	W =   -44.397 deg,	P =     8.168 deg,	R =    14.048 deg
   GP2:
	UF : 1, UT : 1,
	J1=    90.000 deg,	J2=   -90.000 deg
};
P[588]{
   GP1:
	UF : 1, UT : 1,		CONFIG : 'N U T, 0, 0, 0',
	X =  2413.075  mm,	Y =    96.166  mm,	Z =    -3.839  mm,
	W =   -44.394 deg,	P =     8.166 deg,	R =    14.048 deg
   GP2:
	UF : 1, UT : 1,
	J1=    90.000 deg,	J2=   -90.000 deg
};
P[589]{
   GP1:
	UF : 1, UT : 1,		CONFIG : 'N U T, 0, 0, 0',
	X =  1890.253  mm,	Y =  -197.333  mm,	Z =   104.046  mm,
	W =    40.690 deg,	P =   -21.162 deg,	R =    -6.795 deg
   GP2:
	UF : 1, UT : 1,
	J1=    90.000 deg,	J2=   -90.000 deg
};
P[590]{
   GP1:
	UF : 1, UT : 1,		CONFIG : 'N U T, 0, 0, 0',
	X =  1890.254  mm,	Y =  -197.333  mm,	Z =   104.046  mm,
	W =   -33.760 deg,	P =   -16.746 deg,	R =    41.760 deg
   GP2:
	UF : 1, UT : 1,
	J1=    90.000 deg,	J2=   -90.000 deg
};
P[591]{
   GP1:
	UF : 1, UT : 1,		CONFIG : 'N U T, 0, 0, 0',
	X =  2024.254  mm,	Y =  -116.333  mm,	Z =   104.046  mm,
	W =   -36.632 deg,	P =    -7.222 deg,	R =    55.482 deg
   GP2:
	UF : 1, UT : 1,
	J1=    90.000 deg,	J2=   -90.000 deg
};
P[592]{
   GP1:
	UF : 1, UT : 1,		CONFIG : 'N U T, 0, 0, 0',
	X =  2427.383  mm,	Y =    97.382  mm,	Z =     -.048  mm,
	W =   -44.529 deg,	P =    -7.125 deg,	R =    33.229 deg
   GP2:
	UF : 1, UT : 1,
	J1=    90.000 deg,	J2=   -90.000 deg
};
P[593]{
   GP1:
	UF : 1, UT : 1,		CONFIG : 'N U T, 0, 0, 0',
	X =  2337.427  mm,	Y =    71.440  mm,	Z =   847.749  mm,
	W =    45.399 deg,	P =    17.266 deg,	R =    -1.541 deg
   GP2:
	UF : 1, UT : 1,
	J1=    90.000 deg,	J2=   -90.000 deg
};
P[594]{
   GP1:
	UF : 1, UT : 1,		CONFIG : 'N U T, 0, 0, 0',
	X =  2402.831  mm,	Y =   104.785  mm,	Z =   847.602  mm,
	W =    45.390 deg,	P =    17.268 deg,	R =    -1.529 deg
   GP2:
	UF : 1, UT : 1,
	J1=    90.000 deg,	J2=   -90.000 deg
};
P[595]{
   GP1:
	UF : 1, UT : 1,		CONFIG : 'N U T, 0, 0, 0',
	X =  2056.301  mm,	Y =   -98.366  mm,	Z =    49.506  mm,
	W =   -42.382 deg,	P =     2.305 deg,	R =   105.198 deg
   GP2:
	UF : 1, UT : 1,
	J1=    90.000 deg,	J2=   -90.000 deg
};
P[596]{
   GP1:
	UF : 1, UT : 1,		CONFIG : 'N U T, 0, 0, 1',
	X =  1663.323  mm,	Y =  -387.368  mm,	Z =   408.939  mm,
	W =   -27.547 deg,	P =    30.353 deg,	R =   152.229 deg
   GP2:
	UF : 1, UT : 1,
	J1=    90.000 deg,	J2=   -90.000 deg
};
P[597]{
   GP1:
	UF : 1, UT : 1,		CONFIG : 'N U T, 0, 0, 1',
	X =  1656.330  mm,	Y =  -300.541  mm,	Z =  1123.310  mm,
	W =    -7.423 deg,	P =    33.575 deg,	R =  -172.195 deg
   GP2:
	UF : 1, UT : 1,
	J1=    90.000 deg,	J2=   -90.000 deg
};
P[598]{
   GP1:
	UF : 1, UT : 1,		CONFIG : 'N U T, 0, 0, 1',
	X =  2106.086  mm,	Y =  -147.825  mm,	Z =   986.847  mm,
	W =    -2.744 deg,	P =    30.268 deg,	R =  -167.022 deg
   GP2:
	UF : 1, UT : 1,
	J1=    90.000 deg,	J2=   -90.000 deg
};
P[599]{
   GP1:
	UF : 1, UT : 1,		CONFIG : 'N U T, 0, 0, 0',
	X =  2402.842  mm,	Y =   109.949  mm,	Z =   847.942  mm,
	W =     1.452 deg,	P =    40.371 deg,	R =    26.792 deg
   GP2:
	UF : 1, UT : 1,
	J1=    90.000 deg,	J2=   -90.000 deg
};
P[600]{
   GP1:
	UF : 1, UT : 1,		CONFIG : 'N U T, 0, 0, 0',
	X =  2392.403  mm,	Y =   126.094  mm,	Z =   845.932  mm,
	W =     1.448 deg,	P =    40.368 deg,	R =    26.765 deg
   GP2:
	UF : 1, UT : 1,
	J1=    90.000 deg,	J2=   -90.000 deg
};
P[601]{
   GP1:
	UF : 1, UT : 1,		CONFIG : 'F U T, 0, 0, 0',
	X =  2325.472  mm,	Y =    92.116  mm,	Z =   847.036  mm,
	W =   -46.230 deg,	P =   -25.147 deg,	R =    34.050 deg
   GP2:
	UF : 1, UT : 1,
	J1=    90.000 deg,	J2=   -90.000 deg
};
P[602]{
   GP1:
	UF : 1, UT : 1,		CONFIG : 'F U T, 0, 0, 0',
	X =  2391.645  mm,	Y =   126.896  mm,	Z =   847.777  mm,
	W =   -46.222 deg,	P =   -25.150 deg,	R =    34.042 deg
   GP2:
	UF : 1, UT : 1,
	J1=    90.000 deg,	J2=   -90.000 deg
};
P[603]{
   GP1:
	UF : 1, UT : 1,		CONFIG : 'N U T, 0, 0, 0',
	X =  2011.750  mm,	Y =   -80.950  mm,	Z =    -4.575  mm,
	W =    40.372 deg,	P =    23.935 deg,	R =    74.339 deg
   GP2:
	UF : 1, UT : 1,
	J1=    90.000 deg,	J2=  -100.000 deg
};
P[604]{
   GP1:
	UF : 1, UT : 1,		CONFIG : 'N U T, 0, 0, 0',
	X =  2007.194  mm,	Y =   142.177  mm,	Z =   -45.001  mm,
	W =    45.685 deg,	P =     4.509 deg,	R =    78.826 deg
   GP2:
	UF : 1, UT : 1,
	J1=    90.000 deg,	J2=  -100.000 deg
};
P[605]{
   GP1:
	UF : 1, UT : 1,		CONFIG : 'N U T, 0, 0, 0',
	X =  2229.070  mm,	Y =   -48.871  mm,	Z =     4.516  mm,
	W =    44.904 deg,	P =    -3.411 deg,	R =     3.413 deg
   GP2:
	UF : 1, UT : 1,
	J1=    90.000 deg,	J2=   -90.000 deg
};
P[606]{
   GP1:
	UF : 1, UT : 1,		CONFIG : 'N U T, 0, 0, 0',
	X =  2266.341  mm,	Y =   -46.762  mm,	Z =     3.253  mm,
	W =    44.893 deg,	P =    -3.421 deg,	R =     3.427 deg
   GP2:
	UF : 1, UT : 1,
	J1=    90.000 deg,	J2=   -90.000 deg
};
P[607]{
   GP1:
	UF : 1, UT : 1,		CONFIG : 'N U T, 0, 0, 0',
	X =  2096.605  mm,	Y =  -181.583  mm,	Z =   897.867  mm,
	W =     -.064 deg,	P =    31.734 deg,	R =  -164.129 deg
   GP2:
	UF : 1, UT : 1,
	J1=    90.000 deg,	J2=   -90.000 deg
};
P[608]{
   GP1:
	UF : 1, UT : 1,		CONFIG : 'N U T, 0, 0, 0',
	X =  2114.149  mm,	Y =  -253.336  mm,	Z =   921.197  mm,
	W =     1.157 deg,	P =    35.359 deg,	R =   -90.786 deg
   GP2:
	UF : 1, UT : 1,
	J1=    90.000 deg,	J2=   -90.000 deg
};
P[609]{
   GP1:
	UF : 1, UT : 1,		CONFIG : 'N U T, 0, 0, 0',
	X =  2142.334  mm,	Y =   -48.860  mm,	Z =    -3.830  mm,
	W =    44.883 deg,	P =     3.632 deg,	R =    -4.928 deg
   GP2:
	UF : 1, UT : 1,
	J1=    90.000 deg,	J2=   -90.000 deg
};
P[610]{
   GP1:
	UF : 1, UT : 1,		CONFIG : 'N U T, 0, 0, 0',
	X =  2212.734  mm,	Y =   -47.597  mm,	Z =    -4.519  mm,
	W =    44.886 deg,	P =     3.634 deg,	R =    -4.918 deg
   GP2:
	UF : 1, UT : 1,
	J1=    90.000 deg,	J2=   -90.000 deg
};
P[611]{
   GP1:
	UF : 1, UT : 1,		CONFIG : 'N U T, 0, 0, 0',
	X =  2216.176  mm,	Y =   -46.694  mm,	Z =    -5.378  mm,
	W =    44.882 deg,	P =     3.630 deg,	R =   -11.556 deg
   GP2:
	UF : 1, UT : 1,
	J1=    90.000 deg,	J2=   -90.000 deg
};
P[612]{
   GP1:
	UF : 1, UT : 1,		CONFIG : 'N U T, 0, 0, 0',
	X =  1992.932  mm,	Y =   -47.776  mm,	Z =   -14.567  mm,
	W =    44.891 deg,	P =     3.636 deg,	R =    -8.860 deg
   GP2:
	UF : 1, UT : 1,
	J1=    90.000 deg,	J2=   -90.000 deg
};
P[613]{
   GP1:
	UF : 1, UT : 1,		CONFIG : 'N U T, 0, 0, 0',
	X =  2106.099  mm,	Y =   -46.333  mm,	Z =   -15.544  mm,
	W =    44.875 deg,	P =     3.623 deg,	R =    -8.839 deg
   GP2:
	UF : 1, UT : 1,
	J1=    90.000 deg,	J2=   -90.000 deg
};
P[614]{
   GP1:
	UF : 1, UT : 1,		CONFIG : 'N U T, 0, 0, 0',
	X =  2117.103  mm,	Y =   -50.973  mm,	Z =   -11.238  mm,
	W =    41.211 deg,	P =   -19.950 deg,	R =    -8.037 deg
   GP2:
	UF : 1, UT : 1,
	J1=    90.000 deg,	J2=   -90.000 deg
};
P[615]{
   GP1:
	UF : 1, UT : 1,		CONFIG : 'N U T, 0, 0, 0',
	X =  2075.732  mm,	Y =  -109.868  mm,	Z =   -15.932  mm,
	W =   -37.504 deg,	P =      .971 deg,	R =    76.657 deg
   GP2:
	UF : 1, UT : 1,
	J1=    90.000 deg,	J2=   -90.000 deg
};
P[616]{
   GP1:
	UF : 1, UT : 1,		CONFIG : 'N U T, 0, 0, 0',
	X =  2112.001  mm,	Y =   -75.797  mm,	Z =   -17.252  mm,
	W =   -37.498 deg,	P =      .974 deg,	R =    85.226 deg
   GP2:
	UF : 1, UT : 1,
	J1=    90.000 deg,	J2=   -90.000 deg
};
P[617]{
   GP1:
	UF : 1, UT : 1,		CONFIG : 'N U T, 0, 0, 0',
	X =  2126.497  mm,	Y =   -60.152  mm,	Z =   -12.916  mm,
	W =   -48.237 deg,	P =     4.570 deg,	R =   105.632 deg
   GP2:
	UF : 1, UT : 1,
	J1=    89.995 deg,	J2=   -90.001 deg
};
P[618]{
   GP1:
	UF : 1, UT : 1,		CONFIG : 'N U T, 0, 0, 0',
	X =  2628.655  mm,	Y =   126.905  mm,	Z =   907.127  mm,
	W =    31.997 deg,	P =    23.849 deg,	R =   -38.788 deg
   GP2:
	UF : 1, UT : 1,
	J1=    90.000 deg,	J2=   -90.000 deg
};
P[619]{
   GP1:
	UF : 1, UT : 1,		CONFIG : 'N U T, 0, 0, 0',
	X =   949.417  mm,	Y =    74.708  mm,	Z =  1003.698  mm,
	W =    14.657 deg,	P =    21.488 deg,	R =   -36.321 deg
   GP2:
	UF : 1, UT : 1,
	J1=    90.000 deg,	J2=   -90.000 deg
};
P[620]{
   GP1:
	UF : 1, UT : 1,		CONFIG : 'N U T, 0, 0, 0',
	X =   931.440  mm,	Y =   198.476  mm,	Z =   335.127  mm,
	W =   -34.527 deg,	P =    19.136 deg,	R =    25.896 deg
   GP2:
	UF : 1, UT : 1,
	J1=    90.000 deg,	J2=   -90.000 deg
};
P[621]{
   GP1:
	UF : 1, UT : 1,		CONFIG : 'N U T, 0, 0, 0',
	X =  1700.688  mm,	Y =   121.333  mm,	Z =   177.127  mm,
	W =   -48.737 deg,	P =     8.784 deg,	R =     7.978 deg
   GP2:
	UF : 1, UT : 1,
	J1=    90.000 deg,	J2=   -90.000 deg
};
P[622]{
   GP1:
	UF : 1, UT : 1,		CONFIG : 'N U T, 0, 0, 1',
	X =  2137.360  mm,	Y =  -144.268  mm,	Z =   834.187  mm,
	W =      .668 deg,	P =    41.811 deg,	R =  -160.738 deg
   GP2:
	UF : 1, UT : 1,
	J1=    90.000 deg,	J2=   -90.000 deg
};
P[623]{
   GP1:
	UF : 1, UT : 1,		CONFIG : 'N U T, 0, 0, 1',
	X =  2144.152  mm,	Y =  -167.358  mm,	Z =   834.668  mm,
	W =      .532 deg,	P =    40.619 deg,	R =  -160.815 deg
   GP2:
	UF : 1, UT : 1,
	J1=    90.000 deg,	J2=   -90.000 deg
};
P[624]{
   GP1:
	UF : 1, UT : 1,		CONFIG : 'N U T, 0, 0, 0',
	X =  2131.457  mm,	Y =  -193.376  mm,	Z =   832.812  mm,
	W =    -1.789 deg,	P =    43.352 deg,	R =   109.759 deg
   GP2:
	UF : 1, UT : 1,
	J1=    90.000 deg,	J2=   -90.000 deg
};
P[625]{
   GP1:
	UF : 1, UT : 1,		CONFIG : 'N U T, 0, 0, 0',
	X =  2099.029  mm,	Y =  -181.626  mm,	Z =   831.918  mm,
	W =      .955 deg,	P =    43.489 deg,	R =    21.015 deg
   GP2:
	UF : 1, UT : 1,
	J1=    90.000 deg,	J2=   -90.000 deg
};
P[626]{
   GP1:
	UF : 1, UT : 1,		CONFIG : 'N U T, 0, 0, 0',
	X =  1922.982  mm,	Y =    80.524  mm,	Z =   163.198  mm,
	W =   -51.903 deg,	P =     9.364 deg,	R =    21.482 deg
   GP2:
	UF : 1, UT : 1,
	J1=    90.000 deg,	J2=   -90.000 deg
};
P[627]{
   GP1:
	UF : 1, UT : 1,		CONFIG : 'N U T, 0, 0, 0',
	X =  2179.982  mm,	Y =    80.524  mm,	Z =   163.199  mm,
	W =   -51.227 deg,	P =   -13.564 deg,	R =     3.543 deg
   GP2:
	UF : 1, UT : 1,
	J1=    90.000 deg,	J2=   -90.000 deg
};
P[628]{
   GP1:
	UF : 1, UT : 1,		CONFIG : 'N U T, 0, 0, 0',
	X =  2085.167  mm,	Y =  -135.110  mm,	Z =   833.287  mm,
	W =      .566 deg,	P =    42.530 deg,	R =    14.578 deg
   GP2:
	UF : 1, UT : 1,
	J1=    90.000 deg,	J2=   -90.000 deg
};
P[629]{
   GP1:
	UF : 1, UT : 1,		CONFIG : 'N U T, 0, 0, 0',
	X =  2104.005  mm,	Y =  -110.952  mm,	Z =   833.109  mm,
	W =      .858 deg,	P =    43.011 deg,	R =   -74.577 deg
   GP2:
	UF : 1, UT : 1,
	J1=    90.000 deg,	J2=   -90.000 deg
};
P[630]{
   GP1:
	UF : 1, UT : 1,		CONFIG : 'N U T, 0, 0, 0',
	X =  2179.963  mm,	Y =     8.530  mm,	Z =    59.476  mm,
	W =   -44.735 deg,	P =    -5.491 deg,	R =    -5.516 deg
   GP2:
	UF : 1, UT : 1,
	J1=    90.000 deg,	J2=   -90.000 deg
};
P[631]{
   GP1:
	UF : 1, UT : 1,		CONFIG : 'N U T, 0, 0, 0',
	X =  2131.832  mm,	Y =  -123.512  mm,	Z =   834.193  mm,
	W =      .102 deg,	P =    42.115 deg,	R =  -162.102 deg
   GP2:
	UF : 1, UT : 1,
	J1=    90.000 deg,	J2=   -90.000 deg
};
P[632]{
   GP1:
	UF : 1, UT : 1,		CONFIG : 'N U T, 0, 0, 0',
	X =  2138.893  mm,	Y =  -144.672  mm,	Z =   833.681  mm,
	W =      .505 deg,	P =    42.850 deg,	R =  -163.809 deg
   GP2:
	UF : 1, UT : 1,
	J1=    90.000 deg,	J2=   -90.000 deg
};
P[633]{
   GP1:
	UF : 1, UT : 1,		CONFIG : 'N U T, 0, 0, 0',
	X =  2107.700  mm,	Y =  -213.626  mm,	Z =   831.846  mm,
	W =     -.446 deg,	P =    39.556 deg,	R =   -90.694 deg
   GP2:
	UF : 1, UT : 1,
	J1=    90.000 deg,	J2=   -90.000 deg
};
P[634]{
   GP1:
	UF : 1, UT : 1,		CONFIG : 'N U T, 0, 0, 0',
	X =  2083.048  mm,	Y =     5.303  mm,	Z =    47.541  mm,
	W =   -44.735 deg,	P =    -5.491 deg,	R =    -5.516 deg
   GP2:
	UF : 1, UT : 1,
	J1=    90.000 deg,	J2=   -90.000 deg
};
P[635]{
   GP1:
	UF : 1, UT : 1,		CONFIG : 'N U T, 0, 0, 0',
	X =  2200.131  mm,	Y =  -214.897  mm,	Z =   833.980  mm,
	W =     -.446 deg,	P =    39.557 deg,	R =   -90.713 deg
   GP2:
	UF : 1, UT : 1,
	J1=    90.000 deg,	J2=   -90.000 deg
};
P[636]{
   GP1:
	UF : 1, UT : 1,		CONFIG : 'N U T, 0, 0, 0',
	X =  2212.289  mm,	Y =  -210.992  mm,	Z =   834.347  mm,
	W =     -.442 deg,	P =    39.558 deg,	R =   -57.815 deg
   GP2:
	UF : 1, UT : 1,
	J1=    90.000 deg,	J2=   -90.000 deg
};
P[637]{
   GP1:
	UF : 1, UT : 1,		CONFIG : 'N U T, 0, 0, 0',
	X =  2220.486  mm,	Y =  -200.207  mm,	Z =   832.598  mm,
	W =     -.448 deg,	P =    39.556 deg,	R =   -44.056 deg
   GP2:
	UF : 1, UT : 1,
	J1=    90.000 deg,	J2=   -90.000 deg
};
P[638]{
   GP1:
	UF : 1, UT : 1,		CONFIG : 'N U T, 0, 0, 0',
	X =  2065.479  mm,	Y =    84.939  mm,	Z =   110.355  mm,
	W =   -44.734 deg,	P =    -5.490 deg,	R =     4.917 deg
   GP2:
	UF : 1, UT : 1,
	J1=    90.000 deg,	J2=   -90.000 deg
};
P[639]{
   GP1:
	UF : 1, UT : 1,		CONFIG : 'N U T, 0, 0, 0',
	X =  1539.706  mm,	Y = -1470.455  mm,	Z =  1071.063  mm,
	W =   -42.856 deg,	P =   -15.293 deg,	R =    39.131 deg
   GP2:
	UF : 1, UT : 1,
	J1=   180.000 deg,	J2=  -125.000 deg
};
P[640]{
   GP1:
	UF : 1, UT : 1,		CONFIG : 'N U T, 0, 0, 0',
	X =  1166.553  mm,	Y = -1374.013  mm,	Z =  1522.225  mm,
	W =   -32.586 deg,	P =   -12.067 deg,	R =    17.529 deg
   GP2:
	UF : 1, UT : 1,
	J1=   180.000 deg,	J2=  -125.000 deg
};
P[641]{
   GP1:
	UF : 1, UT : 1,		CONFIG : 'N U T, 0, 0, 1',
	X =  1608.479  mm,	Y =   191.940  mm,	Z =    59.355  mm,
	W =    36.994 deg,	P =    27.707 deg,	R =  -122.588 deg
   GP2:
	UF : 1, UT : 1,
	J1=    90.000 deg,	J2=   -90.000 deg
};
P[642]{
   GP1:
	UF : 1, UT : 1,		CONFIG : 'N U T, 0, 0, 0',
	X =  2441.776  mm,	Y =    55.830  mm,	Z =   833.792  mm,
	W =      .117 deg,	P =    42.766 deg,	R =   -42.899 deg
   GP2:
	UF : 1, UT : 1,
	J1=    90.000 deg,	J2=   -90.000 deg
};
P[643]{
   GP1:
	UF : 1, UT : 1,		CONFIG : 'N U T, 0, 0, 0',
	X =  2448.836  mm,	Y =    63.315  mm,	Z =   833.149  mm,
	W =      .109 deg,	P =    42.766 deg,	R =   -49.058 deg
   GP2:
	UF : 1, UT : 1,
	J1=    90.000 deg,	J2=   -90.000 deg
};
P[644]{
   GP1:
	UF : 1, UT : 1,		CONFIG : 'N U T, 0, 0, 0',
	X =  2455.189  mm,	Y =    65.446  mm,	Z =   835.378  mm,
	W =      .109 deg,	P =    42.768 deg,	R =   -56.123 deg
   GP2:
	UF : 1, UT : 1,
	J1=    90.000 deg,	J2=   -90.000 deg
};
P[645]{
   GP1:
	UF : 1, UT : 1,		CONFIG : 'N U T, 0, 0, 0',
	X =  1517.805  mm,	Y =    56.341  mm,	Z =   141.822  mm,
	W =    36.993 deg,	P =    27.706 deg,	R =  -154.189 deg
   GP2:
	UF : 1, UT : 1,
	J1=    90.000 deg,	J2=   -90.000 deg
};
P[646]{
   GP1:
	UF : 1, UT : 1,		CONFIG : 'N U T, 0, 0, 0',
	X =  1476.806  mm,	Y =   169.341  mm,	Z =   386.823  mm,
	W =    23.939 deg,	P =    39.314 deg,	R =  -177.488 deg
   GP2:
	UF : 1, UT : 1,
	J1=    80.000 deg,	J2=   -90.000 deg
};
P[647]{
   GP1:
	UF : 1, UT : 1,		CONFIG : 'N U T, 0, 0, 0',
	X =  2034.807  mm,	Y =   169.341  mm,	Z =   186.823  mm,
	W =    23.939 deg,	P =    39.314 deg,	R =  -177.488 deg
   GP2:
	UF : 1, UT : 1,
	J1=    80.000 deg,	J2=   -90.000 deg
};
P[648]{
   GP1:
	UF : 1, UT : 1,		CONFIG : 'N U T, 0, 0, -1',
	X =  2034.807  mm,	Y =     1.341  mm,	Z =   115.823  mm,
	W =    34.881 deg,	P =    30.459 deg,	R =  -142.693 deg
   GP2:
	UF : 1, UT : 1,
	J1=    80.000 deg,	J2=   -90.000 deg
};
P[649]{
   GP1:
	UF : 1, UT : 1,		CONFIG : 'N U T, 0, 0, 0',
	X =  2645.172  mm,	Y =   206.772  mm,	Z =   838.084  mm,
	W =    29.497 deg,	P =    29.459 deg,	R =    -6.841 deg
   GP2:
	UF : 1, UT : 1,
	J1=    90.000 deg,	J2=   -90.000 deg
};
P[650]{
   GP1:
	UF : 1, UT : 1,		CONFIG : 'N U T, 0, 0, 0',
	X =  2652.713  mm,	Y =   210.527  mm,	Z =   838.644  mm,
	W =    29.493 deg,	P =    29.463 deg,	R =    -6.844 deg
   GP2:
	UF : 1, UT : 1,
	J1=    90.000 deg,	J2=   -90.000 deg
};
P[651]{
   GP1:
	UF : 1, UT : 1,		CONFIG : 'N U T, 0, 0, 0',
	X =  1967.929  mm,	Y =   -36.946  mm,	Z =    54.617  mm,
	W =   -51.899 deg,	P =     9.369 deg,	R =    14.299 deg
   GP2:
	UF : 1, UT : 1,
	J1=    90.000 deg,	J2=   -90.000 deg
};
P[652]{
   GP1:
	UF : 1, UT : 1,		CONFIG : 'N U T, 0, 0, 0',
	X =  1952.806  mm,	Y =   -38.944  mm,	Z =    52.063  mm,
	W =   -51.882 deg,	P =     9.361 deg,	R =     5.846 deg
   GP2:
	UF : 1, UT : 1,
	J1=    90.000 deg,	J2=   -90.000 deg
};
P[653]{
   GP1:
	UF : 1, UT : 1,		CONFIG : 'N U T, 0, 0, 0',
	X =  1695.004  mm,	Y =   -37.169  mm,	Z =    53.060  mm,
	W =   -51.893 deg,	P =     9.370 deg,	R =     5.849 deg
   GP2:
	UF : 1, UT : 1,
	J1=    90.000 deg,	J2=   -90.000 deg
};
P[654]{
   GP1:
	UF : 1, UT : 1,		CONFIG : 'N U T, 0, 0, 0',
	X =  1671.652  mm,	Y =   -33.229  mm,	Z =    53.086  mm,
	W =   -51.882 deg,	P =     9.363 deg,	R =   -32.598 deg
   GP2:
	UF : 1, UT : 1,
	J1=    90.000 deg,	J2=   -90.000 deg
};
P[655]{
   GP1:
	UF : 1, UT : 1,		CONFIG : 'N U T, 0, 0, 0',
	X =  2229.154  mm,	Y =   -35.668  mm,	Z =      .956  mm,
	W =   -45.065 deg,	P =    -5.945 deg,	R =    -3.251 deg
   GP2:
	UF : 1, UT : 1,
	J1=    90.000 deg,	J2=   -90.000 deg
};
P[656]{
   GP1:
	UF : 1, UT : 1,		CONFIG : 'N U T, 0, 0, 0',
	X =  2263.854  mm,	Y =   -39.114  mm,	Z =    -2.230  mm,
	W =   -45.063 deg,	P =    -5.945 deg,	R =    -3.254 deg
   GP2:
	UF : 1, UT : 1,
	J1=    90.000 deg,	J2=   -90.000 deg
};
P[657]{
   GP1:
	UF : 1, UT : 1,		CONFIG : 'N U T, 0, 0, 0',
	X =  2143.762  mm,	Y =   -38.233  mm,	Z =    -9.450  mm,
	W =   -46.267 deg,	P =    -5.650 deg,	R =    -4.455 deg
   GP2:
	UF : 1, UT : 1,
	J1=    89.999 deg,	J2=   -90.000 deg
};
P[658]{
   GP1:
	UF : 1, UT : 1,		CONFIG : 'N U T, 0, 0, 0',
	X =  2211.456  mm,	Y =   -38.697  mm,	Z =   -10.423  mm,
	W =   -44.729 deg,	P =    -5.487 deg,	R =    -5.519 deg
   GP2:
	UF : 1, UT : 1,
	J1=    90.000 deg,	J2=   -90.000 deg
};
P[659]{
   GP1:
	UF : 1, UT : 1,		CONFIG : 'N U T, 0, 0, 0',
	X =  2213.501  mm,	Y =   -38.329  mm,	Z =    -9.533  mm,
	W =   -44.727 deg,	P =    -5.491 deg,	R =    10.507 deg
   GP2:
	UF : 1, UT : 1,
	J1=    90.000 deg,	J2=   -90.000 deg
};
P[660]{
   GP1:
	UF : 1, UT : 1,		CONFIG : 'N U T, 0, 0, 0',
	X =  2115.187  mm,	Y =   -36.549  mm,	Z =   -16.802  mm,
	W =   -44.729 deg,	P =    -5.491 deg,	R =    -5.515 deg
   GP2:
	UF : 1, UT : 1,
	J1=    90.000 deg,	J2=   -90.000 deg
};
P[661]{
   GP1:
	UF : 1, UT : 1,		CONFIG : 'N U T, 0, 0, 0',
	X =  2031.075  mm,	Y =   -35.591  mm,	Z =   -15.945  mm,
	W =   -44.726 deg,	P =    -5.493 deg,	R =    -5.522 deg
   GP2:
	UF : 1, UT : 1,
	J1=    90.000 deg,	J2=   -90.000 deg
};
P[662]{
   GP1:
	UF : 1, UT : 1,		CONFIG : 'N U T, 0, 0, 0',
	X =  2012.774  mm,	Y =   -33.603  mm,	Z =   -16.255  mm,
	W =   -44.728 deg,	P =    -5.488 deg,	R =   -41.543 deg
   GP2:
	UF : 1, UT : 1,
	J1=    90.000 deg,	J2=   -90.000 deg
};
P[663]{
   GP1:
	UF : 1, UT : 1,		CONFIG : 'N U T, 0, 0, 0',
	X =  1659.349  mm,	Y =   229.576  mm,	Z =   -15.827  mm,
	W =    34.860 deg,	P =    26.474 deg,	R =  -126.851 deg
   GP2:
	UF : 1, UT : 1,
	J1=    90.000 deg,	J2=   -90.000 deg
};
P[664]{
   GP1:
	UF : 1, UT : 1,		CONFIG : 'N U T, 0, 0, 1',
	X =  1662.403  mm,	Y =    10.748  mm,	Z =   -16.240  mm,
	W =    36.966 deg,	P =    27.691 deg,	R =  -122.597 deg
   GP2:
	UF : 1, UT : 1,
	J1=    90.000 deg,	J2=   -90.000 deg
};
P[665]{
   GP1:
	UF : 1, UT : 1,		CONFIG : 'N U T, 0, 0, 0',
	X =  1661.230  mm,	Y =   -12.152  mm,	Z =   -15.927  mm,
	W =    37.079 deg,	P =    27.798 deg,	R =  -137.823 deg
   GP2:
	UF : 1, UT : 1,
	J1=    90.000 deg,	J2=   -90.000 deg
};
P[666]{
   GP1:
	UF : 1, UT : 1,		CONFIG : 'N U T, 0, 0, 0',
	X =  2070.256  mm,	Y =   -29.016  mm,	Z =    17.551  mm,
	W =    27.122 deg,	P =    24.041 deg,	R =  -162.981 deg
   GP2:
	UF : 1, UT : 1,
	J1=    80.000 deg,	J2=   -90.000 deg
};
P[667]{
   GP1:
	UF : 1, UT : 1,		CONFIG : 'N U T, 0, 0, 1',
	X =  2077.472  mm,	Y =     9.268  mm,	Z =    15.852  mm,
	W =    26.540 deg,	P =    23.907 deg,	R =  -139.393 deg
   GP2:
	UF : 1, UT : 1,
	J1=    80.000 deg,	J2=   -90.000 deg
};
P[668]{
   GP1:
	UF : 1, UT : 1,		CONFIG : 'N U T, 0, 0, 0',
	X =  2079.821  mm,	Y =    18.267  mm,	Z =    15.557  mm,
	W =    26.544 deg,	P =    23.915 deg,	R =  -163.856 deg
   GP2:
	UF : 1, UT : 1,
	J1=    80.000 deg,	J2=   -90.000 deg
};
P[669]{
   GP1:
	UF : 1, UT : 1,		CONFIG : 'N U T, 0, 0, 0',
	X =  2088.621  mm,	Y =    27.690  mm,	Z =    13.857  mm,
	W =    17.944 deg,	P =    33.024 deg,	R =   153.337 deg
   GP2:
	UF : 1, UT : 1,
	J1=    80.000 deg,	J2=   -90.000 deg
};
P[670]{
   GP1:
	UF : 1, UT : 1,		CONFIG : 'N U T, 0, 0, 0',
	X =  2492.536  mm,	Y =   739.403  mm,	Z =    25.184  mm,
	W =   -42.166 deg,	P =     5.515 deg,	R =   107.587 deg
   GP2:
	UF : 1, UT : 1,
	J1=    80.000 deg,	J2=   -90.000 deg
};
P[671]{
   GP1:
	UF : 1, UT : 1,		CONFIG : 'N U T, 0, 0, 0',
	X =  2492.536  mm,	Y =   809.403  mm,	Z =    25.184  mm,
	W =   -35.462 deg,	P =    25.069 deg,	R =   132.276 deg
   GP2:
	UF : 1, UT : 1,
	J1=    80.000 deg,	J2=   -90.000 deg
};
P[672]{
   GP1:
	UF : 1, UT : 1,		CONFIG : 'N U T, 0, 0, 0',
	X =  2236.640  mm,	Y =   176.401  mm,	Z =    -7.067  mm,
	W =     2.794 deg,	P =    36.171 deg,	R =   129.508 deg
   GP2:
	UF : 1, UT : 1,
	J1=    80.000 deg,	J2=   -90.000 deg
};
P[673]{
   GP1:
	UF : 1, UT : 1,		CONFIG : 'N U T, 0, 0, 0',
	X =  2264.963  mm,	Y =   203.116  mm,	Z =   -13.114  mm,
	W =     3.306 deg,	P =    33.869 deg,	R =   124.421 deg
   GP2:
	UF : 1, UT : 1,
	J1=    80.000 deg,	J2=   -90.000 deg
};
P[674]{
   GP1:
	UF : 1, UT : 1,		CONFIG : 'N U T, 0, 0, 0',
	X =  2287.031  mm,	Y =   217.729  mm,	Z =   -16.695  mm,
	W =     6.006 deg,	P =    35.930 deg,	R =   123.381 deg
   GP2:
	UF : 1, UT : 1,
	J1=    80.000 deg,	J2=   -90.000 deg
};
P[675]{
   GP1:
	UF : 1, UT : 1,		CONFIG : 'N U T, 0, 0, 0',
	X =  2387.696  mm,	Y =   277.952  mm,	Z =   -35.568  mm,
	W =     8.794 deg,	P =    37.204 deg,	R =   129.070 deg
   GP2:
	UF : 1, UT : 1,
	J1=    80.000 deg,	J2=   -90.000 deg
};
P[676]{
   GP1:
	UF : 1, UT : 1,		CONFIG : 'N U T, 0, 0, 0',
	X =  2404.670  mm,	Y =   288.506  mm,	Z =   -40.636  mm,
	W =    -2.498 deg,	P =    34.190 deg,	R =   123.664 deg
   GP2:
	UF : 1, UT : 1,
	J1=    80.000 deg,	J2=   -90.000 deg
};
P[677]{
   GP1:
	UF : 1, UT : 1,		CONFIG : 'N U T, 0, 0, 0',
	X =  2423.597  mm,	Y =   314.103  mm,	Z =   -39.372  mm,
	W =      .578 deg,	P =    31.082 deg,	R =   135.853 deg
   GP2:
	UF : 1, UT : 1,
	J1=    80.000 deg,	J2=   -90.000 deg
};
P[678]{
   GP1:
	UF : 1, UT : 1,		CONFIG : 'N U T, 0, 0, 0',
	X =  2506.157  mm,	Y =   429.784  mm,	Z =   -53.556  mm,
	W =   -18.684 deg,	P =    29.858 deg,	R =   100.231 deg
   GP2:
	UF : 1, UT : 1,
	J1=    80.000 deg,	J2=   -90.000 deg
};
P[679]{
   GP1:
	UF : 1, UT : 1,		CONFIG : 'N U T, 0, 0, 0',
	X =  2521.799  mm,	Y =   685.855  mm,	Z =   110.598  mm,
	W =   -11.653 deg,	P =   -32.812 deg,	R =    68.201 deg
   GP2:
	UF : 1, UT : 1,
	J1=    80.000 deg,	J2=   -90.000 deg
};
P[680]{
   GP1:
	UF : 1, UT : 1,		CONFIG : 'N U T, 0, 0, 0',
	X =  2352.111  mm,	Y =   297.878  mm,	Z =   188.758  mm,
	W =   -43.260 deg,	P =    61.542 deg,	R =   123.185 deg
   GP2:
	UF : 1, UT : 1,
	J1=    80.000 deg,	J2=   -90.000 deg
};
P[681]{
   GP1:
	UF : 1, UT : 1,		CONFIG : 'N U T, 0, 0, 0',
	X =  1368.100  mm,	Y =   306.117  mm,	Z =   479.720  mm,
	W =   -45.599 deg,	P =    57.111 deg,	R =   114.814 deg
   GP2:
	UF : 1, UT : 1,
	J1=    80.000 deg,	J2=   -90.000 deg
};
P[682]{
   GP1:
	UF : 1, UT : 1,		CONFIG : 'N U B, 0, 0, 0',
	X =   356.032  mm,	Y =    -2.146  mm,	Z =  2424.049  mm,
	W =      .001 deg,	P =   -40.002 deg,	R =     -.005 deg
   GP2:
	UF : 1, UT : 1,
	J1=   180.000 deg,	J2=  -150.000 deg
};
P[683]{
   GP1:
	UF : 1, UT : 1,		CONFIG : 'N U T, 0, 0, 0',
	X =   642.423  mm,	Y = -1094.246  mm,	Z =  1725.795  mm,
	W =     2.647 deg,	P =   -31.291 deg,	R =   -11.601 deg
   GP2:
	UF : 1, UT : 1,
	J1=   180.000 deg,	J2=  -150.000 deg
};
P[684]{
   GP1:
	UF : 1, UT : 1,		CONFIG : 'N U T, 0, 0, 0',
	X =   799.244  mm,	Y = -1202.971  mm,	Z =  1035.322  mm,
	W =    24.190 deg,	P =   -39.178 deg,	R =    -6.255 deg
   GP2:
	UF : 1, UT : 1,
	J1=   180.000 deg,	J2=  -150.000 deg
};
P[685]{
   GP1:
	UF : 1, UT : 1,		CONFIG : 'N U T, 0, 0, 0',
	X =   954.244  mm,	Y = -1102.971  mm,	Z =   861.322  mm,
	W =    24.190 deg,	P =   -39.178 deg,	R =    -6.255 deg
   GP2:
	UF : 1, UT : 1,
	J1=   180.000 deg,	J2=  -150.000 deg
};
P[686]{
   GP1:
	UF : 1, UT : 1,		CONFIG : 'N U T, 0, 0, 0',
	X =  2522.874  mm,	Y =   447.428  mm,	Z =   -56.211  mm,
	W =   -18.818 deg,	P =    32.562 deg,	R =    79.861 deg
   GP2:
	UF : 1, UT : 1,
	J1=    80.000 deg,	J2=   -90.000 deg
};
P[687]{
   GP1:
	UF : 1, UT : 1,		CONFIG : 'N U T, 0, 0, 0',
	X =  2554.598  mm,	Y =   458.467  mm,	Z =   -62.590  mm,
	W =   -16.507 deg,	P =    33.838 deg,	R =    74.968 deg
   GP2:
	UF : 1, UT : 1,
	J1=    80.000 deg,	J2=   -90.000 deg
};
P[688]{
   GP1:
	UF : 1, UT : 1,		CONFIG : 'N U T, 0, 0, 0',
	X =   955.526  mm,	Y = -1174.727  mm,	Z =   902.888  mm,
	W =    27.863 deg,	P =   -46.318 deg,	R =   -16.260 deg
   GP2:
	UF : 1, UT : 1,
	J1=   180.000 deg,	J2=  -150.000 deg
};
P[689]{
   GP1:
	UF : 1, UT : 1,		CONFIG : 'N U T, 0, 0, 0',
	X =   571.093  mm,	Y = -1097.630  mm,	Z =  1035.072  mm,
	W =    42.871 deg,	P =   -15.240 deg,	R =   -45.029 deg
   GP2:
	UF : 1, UT : 1,
	J1=   180.000 deg,	J2=  -150.000 deg
};
P[690]{
   GP1:
	UF : 1, UT : 1,		CONFIG : 'N U T, 0, 0, 0',
	X =   749.093  mm,	Y =  -654.630  mm,	Z =   835.073  mm,
	W =    44.064 deg,	P =   -10.243 deg,	R =   -50.428 deg
   GP2:
	UF : 1, UT : 1,
	J1=   180.000 deg,	J2=  -150.000 deg
};
P[691]{
   GP1:
	UF : 1, UT : 1,		CONFIG : 'N U T, 0, 0, 0',
	X =  2567.108  mm,	Y =   460.127  mm,	Z =   -64.835  mm,
	W =   -16.506 deg,	P =    33.836 deg,	R =    74.958 deg
   GP2:
	UF : 1, UT : 1,
	J1=    80.000 deg,	J2=   -90.000 deg
};
P[692]{
   GP1:
	UF : 1, UT : 1,		CONFIG : 'N U T, 0, 0, 0',
	X =  2609.688  mm,	Y =   486.425  mm,	Z =   -71.766  mm,
	W =   -17.685 deg,	P =    33.469 deg,	R =   110.387 deg
   GP2:
	UF : 1, UT : 1,
	J1=    80.000 deg,	J2=   -90.000 deg
};
P[693]{
   GP1:
	UF : 1, UT : 1,		CONFIG : 'N U T, 0, 0, 0',
	X =  2628.545  mm,	Y =   536.100  mm,	Z =   -75.597  mm,
	W =   -28.178 deg,	P =    11.271 deg,	R =   110.042 deg
   GP2:
	UF : 1, UT : 1,
	J1=    80.000 deg,	J2=   -90.000 deg
};
P[694]{
   GP1:
	UF : 1, UT : 1,		CONFIG : 'N U T, 0, 0, 0',
	X =   962.545  mm,	Y = -1093.036  mm,	Z =   867.966  mm,
	W =    44.863 deg,	P =     3.974 deg,	R =   -63.984 deg
   GP2:
	UF : 1, UT : 1,
	J1=   180.000 deg,	J2=  -150.000 deg
};
P[695]{
   GP1:
	UF : 1, UT : 1,		CONFIG : 'N U T, 0, 0, 0',
	X =   592.698  mm,	Y =  -634.536  mm,	Z =   863.966  mm,
	W =    36.388 deg,	P =   -28.554 deg,	R =   -27.033 deg
   GP2:
	UF : 1, UT : 1,
	J1=   180.000 deg,	J2=  -150.000 deg
};
P[696]{
   GP1:
	UF : 1, UT : 1,		CONFIG : 'N U T, 0, 0, 0',
	X =  2632.222  mm,	Y =   732.009  mm,	Z =   -80.623  mm,
	W =   -28.919 deg,	P =    12.962 deg,	R =   109.016 deg
   GP2:
	UF : 1, UT : 1,
	J1=    80.000 deg,	J2=   -90.000 deg
};
P[697]{
   GP1:
	UF : 1, UT : 1,		CONFIG : 'N U T, 0, 0, 0',
	X =  2634.037  mm,	Y =   736.946  mm,	Z =   -80.036  mm,
	W =   -28.912 deg,	P =    12.964 deg,	R =    86.663 deg
   GP2:
	UF : 1, UT : 1,
	J1=    80.000 deg,	J2=   -90.000 deg
};
P[698]{
   GP1:
	UF : 1, UT : 1,		CONFIG : 'N U T, 0, 0, 0',
	X =   545.804  mm,	Y =  -597.246  mm,	Z =   979.702  mm,
	W =    15.937 deg,	P =   -42.493 deg,	R =     6.853 deg
   GP2:
	UF : 1, UT : 1,
	J1=   180.000 deg,	J2=  -150.000 deg
};
P[699]{
   GP1:
	UF : 1, UT : 1,		CONFIG : 'N U T, 0, 0, 0',
	X =   373.944  mm,	Y =  -794.657  mm,	Z =  1562.528  mm,
	W =    12.204 deg,	P =   -25.221 deg,	R =   -18.478 deg
   GP2:
	UF : 1, UT : 1,
	J1=   180.000 deg,	J2=  -150.000 deg
};
P[700]{
   GP1:
	UF : 1, UT : 1,		CONFIG : 'N U T, 0, 0, 0',
	X =   958.519  mm,	Y =  -942.564  mm,	Z =  1465.461  mm,
	W =     -.010 deg,	P =    45.866 deg,	R =    90.000 deg
   GP2:
	UF : 0, UT : 1,
	J1=   180.000 deg,	J2=   -90.000 deg
};
P[701]{
   GP1:
	UF : 1, UT : 1,		CONFIG : 'N U T, 0, 0, 0',
	X =  1863.519  mm,	Y = -1304.565  mm,	Z =  1265.460  mm,
	W =   -41.810 deg,	P =   -20.894 deg,	R =   -21.724 deg
   GP2:
	UF : 0, UT : 1,
	J1=   180.000 deg,	J2=   -90.000 deg
};
P[702]{
   GP1:
	UF : 1, UT : 1,		CONFIG : 'N U T, 0, 0, 0',
	X =  1929.519  mm,	Y = -1405.565  mm,	Z =  1058.460  mm,
	W =   -42.701 deg,	P =    18.644 deg,	R =    19.122 deg
   GP2:
	UF : 0, UT : 1,
	J1=   180.000 deg,	J2=   -90.000 deg
};
P[703]{
   GP1:
	UF : 1, UT : 1,		CONFIG : 'N U T, 0, 0, 0',
	X =  2636.521  mm,	Y =   741.783  mm,	Z =   -80.114  mm,
	W =   -28.912 deg,	P =    12.964 deg,	R =    81.290 deg
   GP2:
	UF : 1, UT : 1,
	J1=    80.000 deg,	J2=   -90.000 deg
};
P[704]{
   GP1:
	UF : 1, UT : 1,		CONFIG : 'N U T, 0, 0, 0',
	X =  2643.067  mm,	Y =   762.281  mm,	Z =   -80.422  mm,
	W =   -29.832 deg,	P =     9.276 deg,	R =    88.856 deg
   GP2:
	UF : 1, UT : 1,
	J1=    80.000 deg,	J2=   -90.000 deg
};
P[705]{
   GP1:
	UF : 1, UT : 1,		CONFIG : 'N U T, 0, 0, 0',
	X =  2640.869  mm,	Y =   777.391  mm,	Z =   -80.196  mm,
	W =   -33.768 deg,	P =      .740 deg,	R =   112.866 deg
   GP2:
	UF : 1, UT : 1,
	J1=    80.000 deg,	J2=   -90.000 deg
};
P[706]{
   GP1:
	UF : 1, UT : 1,		CONFIG : 'N U T, 0, 0, 0',
	X =  2554.805  mm,	Y =   840.968  mm,	Z =   -65.386  mm,
	W =   -31.195 deg,	P =     9.618 deg,	R =   105.424 deg
   GP2:
	UF : 1, UT : 1,
	J1=    80.000 deg,	J2=   -90.000 deg
};
P[707]{
   GP1:
	UF : 1, UT : 1,		CONFIG : 'N U T, 0, 0, 0',
	X =  2556.195  mm,	Y =   827.922  mm,	Z =   -66.293  mm,
	W =   -32.481 deg,	P =     1.245 deg,	R =    91.949 deg
   GP2:
	UF : 1, UT : 1,
	J1=    80.000 deg,	J2=   -90.000 deg
};
P[708]{
   GP1:
	UF : 1, UT : 1,		CONFIG : 'N U T, 0, 0, 0',
	X =  2039.010  mm,	Y = -1381.508  mm,	Z =  1071.568  mm,
	W =   -44.862 deg,	P =     3.961 deg,	R =   -20.537 deg
   GP2:
	UF : 0, UT : 1,
	J1=   180.000 deg,	J2=   -90.000 deg
};
P[709]{
   GP1:
	UF : 1, UT : 1,		CONFIG : 'N U T, 0, 0, 0',
	X =  2562.628  mm,	Y =   816.135  mm,	Z =   -66.477  mm,
	W =   -29.304 deg,	P =   -14.723 deg,	R =   104.306 deg
   GP2:
	UF : 1, UT : 1,
	J1=    80.000 deg,	J2=   -90.000 deg
};
P[710]{
   GP1:
	UF : 1, UT : 1,		CONFIG : 'N U T, 0, 0, 0',
	X =  1341.730  mm,	Y =  -571.237  mm,	Z =  1990.182  mm,
	W =   -18.602 deg,	P =   -32.070 deg,	R =   -22.859 deg
   GP2:
	UF : 1, UT : 1,
	J1=   180.000 deg,	J2=   -90.000 deg
};
P[711]{
   GP1:
	UF : 1, UT : 1,		CONFIG : 'N U T, 0, 0, 0',
	X =  1392.804  mm,	Y =   640.782  mm,	Z =  1670.105  mm,
	W =    37.735 deg,	P =   -20.539 deg,	R =     -.894 deg
   GP2:
	UF : 0, UT : 1,
	J1=   180.000 deg,	J2=    90.000 deg
};
P[712]{
   GP1:
	UF : 1, UT : 1,		CONFIG : 'N U T, 0, 0, 0',
	X =  1849.519  mm,	Y =  1220.906  mm,	Z =  1351.461  mm,
	W =    44.958 deg,	P =    -2.212 deg,	R =     2.229 deg
   GP2:
	UF : 0, UT : 1,
	J1=   180.000 deg,	J2=    90.000 deg
};
P[713]{
   GP1:
	UF : 1, UT : 1,		CONFIG : 'N U T, 0, 0, 0',
	X =  1880.451  mm,	Y =  1275.016  mm,	Z =  1238.303  mm,
	W =    44.592 deg,	P =     6.805 deg,	R =    -6.838 deg
   GP2:
	UF : 1, UT : 1,
	J1=   180.000 deg,	J2=    90.000 deg
};
P[714]{
   GP1:
	UF : 1, UT : 1,		CONFIG : 'N U T, 0, 0, 0',
	X =  1926.400  mm,	Y =  1355.399  mm,	Z =  1070.204  mm,
	W =    41.277 deg,	P =    19.800 deg,	R =   -21.086 deg
   GP2:
	UF : 0, UT : 1,
	J1=   180.000 deg,	J2=    90.000 deg
};
P[715]{
   GP1:
	UF : 1, UT : 1,		CONFIG : 'N U T, 0, 0, 0',
	X =  2576.087  mm,	Y =   812.043  mm,	Z =   -72.164  mm,
	W =    -3.300 deg,	P =   -34.456 deg,	R =   105.021 deg
   GP2:
	UF : 1, UT : 1,
	J1=    80.000 deg,	J2=   -90.000 deg
};
P[716]{
   GP1:
	UF : 1, UT : 1,		CONFIG : 'N U T, 0, 0, 0',
	X =  2599.271  mm,	Y =   811.663  mm,	Z =   -77.249  mm,
	W =    -3.299 deg,	P =   -34.461 deg,	R =   105.020 deg
   GP2:
	UF : 1, UT : 1,
	J1=    80.000 deg,	J2=   -90.000 deg
};
P[717]{
   GP1:
	UF : 1, UT : 1,		CONFIG : 'N U T, 0, 0, 0',
	X =  2617.323  mm,	Y =   805.644  mm,	Z =   -77.465  mm,
	W =     3.038 deg,	P =   -34.483 deg,	R =    65.938 deg
   GP2:
	UF : 1, UT : 1,
	J1=    80.000 deg,	J2=   -90.000 deg
};
P[718]{
   GP1:
	UF : 1, UT : 1,		CONFIG : 'N U T, 0, 0, 0',
	X =  2640.391  mm,	Y =   775.794  mm,	Z =   -80.773  mm,
	W =   -11.649 deg,	P =   -32.807 deg,	R =    38.714 deg
   GP2:
	UF : 1, UT : 1,
	J1=    80.000 deg,	J2=   -90.000 deg
};
P[719]{
   GP1:
	UF : 1, UT : 1,		CONFIG : 'N U T, 0, 0, 0',
	X =  1063.279  mm,	Y = -1053.306  mm,	Z =   783.332  mm,
	W =    24.557 deg,	P =   -38.977 deg,	R =    -6.176 deg
   GP2:
	UF : 1, UT : 1,
	J1=   180.000 deg,	J2=  -150.000 deg
};
P[720]{
   GP1:
	UF : 1, UT : 1,		CONFIG : 'N U T, 0, 0, 0',
	X =  1993.007  mm,	Y =  1431.170  mm,	Z =  1068.677  mm,
	W =    44.305 deg,	P =     8.850 deg,	R =     3.803 deg
   GP2:
	UF : 1, UT : 1,
	J1=   180.000 deg,	J2=    90.000 deg
};
P[721]{
   GP1:
	UF : 1, UT : 1,		CONFIG : 'N U T, 0, 0, 0',
	X =  1840.948  mm,	Y =  1174.835  mm,	Z =  1330.032  mm,
	W =    44.958 deg,	P =    -2.212 deg,	R =     2.229 deg
   GP2:
	UF : 0, UT : 1,
	J1=   180.000 deg,	J2=    90.000 deg
};
P[722]{
   GP1:
	UF : 1, UT : 1,		CONFIG : 'N U T, 0, 0, 0',
	X =   975.793  mm,	Y =  -256.447  mm,	Z =  2489.902  mm,
	W =   -88.787 deg,	P =   -13.157 deg,	R =    77.737 deg
   GP2:
	UF : 1, UT : 1,
	J1=   100.000 deg,	J2=   -90.000 deg
};
P[723]{
   GP1:
	UF : 1, UT : 1,		CONFIG : 'N U T, 0, 0, 0',
	X =  1109.166  mm,	Y = -1127.961  mm,	Z =   780.009  mm,
	W =    24.527 deg,	P =   -38.988 deg,	R =    -6.133 deg
   GP2:
	UF : 1, UT : 1,
	J1=   180.000 deg,	J2=  -150.000 deg
};
P[724]{
   GP1:
	UF : 1, UT : 1,		CONFIG : 'N U T, 0, 0, 0',
	X =   786.252  mm,	Y =  -573.217  mm,	Z =   780.478  mm,
	W =    38.067 deg,	P =   -23.497 deg,	R =   -32.642 deg
   GP2:
	UF : 1, UT : 1,
	J1=   180.000 deg,	J2=  -150.000 deg
};
P[725]{
   GP1:
	UF : 1, UT : 1,		CONFIG : 'N U T, 0, 0, 0',
	X =   927.792  mm,	Y =  -818.010  mm,	Z =   778.982  mm,
	W =    43.362 deg,	P =    -6.897 deg,	R =   -57.357 deg
   GP2:
	UF : 1, UT : 1,
	J1=   180.000 deg,	J2=  -150.000 deg
};
P[726]{
   GP1:
	UF : 1, UT : 1,		CONFIG : 'N U T, 0, 0, 0',
	X =  1047.239  mm,	Y = -1021.242  mm,	Z =   783.994  mm,
	W =    37.928 deg,	P =   -23.474 deg,	R =   -37.343 deg
   GP2:
	UF : 1, UT : 1,
	J1=   180.000 deg,	J2=  -150.000 deg
};
P[727]{
   GP1:
	UF : 1, UT : 1,		CONFIG : 'N U T, 0, 0, 0',
	X =   765.614  mm,	Y =  -535.452  mm,	Z =   786.067  mm,
	W =    41.849 deg,	P =   -18.077 deg,	R =   -40.922 deg
   GP2:
	UF : 1, UT : 1,
	J1=   180.000 deg,	J2=  -150.000 deg
};
P[728]{
   GP1:
	UF : 1, UT : 1,		CONFIG : 'N U T, 0, 0, 0',
	X =   721.837  mm,	Y =  -462.053  mm,	Z =   783.548  mm,
	W =    27.769 deg,	P =   -36.841 deg,	R =   -11.320 deg
   GP2:
	UF : 1, UT : 1,
	J1=   180.000 deg,	J2=  -150.000 deg
};
P[729]{
   GP1:
	UF : 1, UT : 1,		CONFIG : 'N U T, 0, 0, 0',
	X =  1898.693  mm,	Y = -1465.196  mm,	Z =  1035.174  mm,
	W =   -39.886 deg,	P =    23.861 deg,	R =    23.910 deg
   GP2:
	UF : 1, UT : 1,
	J1=   180.000 deg,	J2=   -90.000 deg
};
P[730]{
   GP1:
	UF : 1, UT : 1,		CONFIG : 'N U T, 0, 0, 0',
	X =  1930.842  mm,	Y = -1465.932  mm,	Z =  1036.894  mm,
	W =   -43.540 deg,	P =    14.560 deg,	R =    14.833 deg
   GP2:
	UF : 1, UT : 1,
	J1=   180.000 deg,	J2=   -90.000 deg
};
P[731]{
   GP1:
	UF : 1, UT : 1,		CONFIG : 'N U T, 0, 0, 0',
	X =  1966.391  mm,	Y = -1464.791  mm,	Z =  1037.270  mm,
	W =   -43.537 deg,	P =    14.558 deg,	R =    14.821 deg
   GP2:
	UF : 1, UT : 1,
	J1=   180.000 deg,	J2=   -90.000 deg
};
P[732]{
   GP1:
	UF : 1, UT : 1,		CONFIG : 'F U T, 0, 0, 0',
	X =   804.374  mm,	Y =   981.069  mm,	Z =  1117.927  mm,
	W =    50.730 deg,	P =      .639 deg,	R =   -51.736 deg
   GP2:
	UF : 1, UT : 1,
	J1=   180.000 deg,	J2=   150.000 deg
};
P[733]{
   GP1:
	UF : 1, UT : 1,		CONFIG : 'F U T, 0, 0, 0',
	X =  1064.016  mm,	Y =   999.283  mm,	Z =  1072.926  mm,
	W =    50.730 deg,	P =      .639 deg,	R =   -51.736 deg
   GP2:
	UF : 1, UT : 1,
	J1=   180.000 deg,	J2=   150.000 deg
};
P[734]{
   GP1:
	UF : 1, UT : 1,		CONFIG : 'N U T, 0, 0, 0',
	X =  1996.744  mm,	Y = -1479.610  mm,	Z =  1035.370  mm,
	W =   -43.544 deg,	P =    14.560 deg,	R =   -14.022 deg
   GP2:
	UF : 1, UT : 1,
	J1=   180.000 deg,	J2=   -90.000 deg
};
P[735]{
   GP1:
	UF : 1, UT : 1,		CONFIG : 'N U T, 0, 0, 0',
	X =  2005.341  mm,	Y = -1493.994  mm,	Z =  1032.872  mm,
	W =   -44.808 deg,	P =     8.522 deg,	R =   -27.704 deg
   GP2:
	UF : 1, UT : 1,
	J1=   180.000 deg,	J2=   -90.000 deg
};
P[736]{
   GP1:
	UF : 1, UT : 1,		CONFIG : 'N U T, 0, 0, 0',
	X =  1897.818  mm,	Y =  1491.288  mm,	Z =  1034.377  mm,
	W =    41.278 deg,	P =    19.806 deg,	R =   -17.231 deg
   GP2:
	UF : 1, UT : 1,
	J1=   180.000 deg,	J2=    90.000 deg
};
P[737]{
   GP1:
	UF : 1, UT : 1,		CONFIG : 'N U T, 0, 0, 0',
	X =  1932.829  mm,	Y =  1488.728  mm,	Z =  1037.568  mm,
	W =    41.270 deg,	P =    19.801 deg,	R =   -17.222 deg
   GP2:
	UF : 1, UT : 1,
	J1=   180.000 deg,	J2=    90.000 deg
};
P[738]{
   GP1:
	UF : 1, UT : 1,		CONFIG : 'F U T, 0, 0, 0',
	X =  1102.958  mm,	Y =   975.094  mm,	Z =  1056.986  mm,
	W =    50.535 deg,	P =   -23.426 deg,	R =   -25.981 deg
   GP2:
	UF : 1, UT : 1,
	J1=   180.000 deg,	J2=   150.000 deg
};
P[739]{
   GP1:
	UF : 1, UT : 1,		CONFIG : 'F U T, 0, 0, 0',
	X =   851.887  mm,	Y =   977.237  mm,	Z =  1067.701  mm,
	W =    50.535 deg,	P =   -23.426 deg,	R =   -25.981 deg
   GP2:
	UF : 1, UT : 1,
	J1=   180.000 deg,	J2=   150.000 deg
};
P[740]{
   GP1:
	UF : 1, UT : 1,		CONFIG : 'F U T, 0, 0, 0',
	X =   626.208  mm,	Y =  1096.450  mm,	Z =  1381.774  mm,
	W =    61.728 deg,	P =   -31.893 deg,	R =   -10.883 deg
   GP2:
	UF : 1, UT : 1,
	J1=   180.000 deg,	J2=   150.000 deg
};
P[741]{
   GP1:
	UF : 1, UT : 1,		CONFIG : 'N U T, 0, 0, 0',
	X =  1964.476  mm,	Y =  1486.706  mm,	Z =  1040.490  mm,
	W =    41.276 deg,	P =    19.802 deg,	R =   -17.225 deg
   GP2:
	UF : 1, UT : 1,
	J1=   180.000 deg,	J2=    90.000 deg
};
P[742]{
   GP1:
	UF : 1, UT : 1,		CONFIG : 'N U T, 0, 0, 0',
	X =  1987.397  mm,	Y =  1501.086  mm,	Z =  1037.179  mm,
	W =    41.274 deg,	P =    19.802 deg,	R =     6.738 deg
   GP2:
	UF : 1, UT : 1,
	J1=   180.000 deg,	J2=    90.000 deg
};
P[743]{
   GP1:
	UF : 1, UT : 1,		CONFIG : 'N U T, 0, 0, 0',
	X =  1995.872  mm,	Y =  1510.585  mm,	Z =  1037.723  mm,
	W =    43.860 deg,	P =    11.269 deg,	R =    16.934 deg
   GP2:
	UF : 1, UT : 1,
	J1=   180.000 deg,	J2=    90.000 deg
};
P[744]{
   GP1:
	UF : 1, UT : 1,		CONFIG : 'N U T, 0, 0, 0',
	X =  1643.566  mm,	Y = -1408.541  mm,	Z =  1035.422  mm,
	W =   -42.856 deg,	P =   -15.294 deg,	R =    39.130 deg
   GP2:
	UF : 1, UT : 1,
	J1=   180.000 deg,	J2=  -125.000 deg
};
P[745]{
   GP1:
	UF : 1, UT : 1,		CONFIG : 'N U T, 0, 0, 0',
	X =  1652.001  mm,	Y = -1400.198  mm,	Z =  1034.064  mm,
	W =   -42.573 deg,	P =   -16.796 deg,	R =    40.474 deg
   GP2:
	UF : 1, UT : 1,
	J1=   180.000 deg,	J2=  -125.000 deg
};
P[746]{
   GP1:
	UF : 1, UT : 1,		CONFIG : 'N U T, 0, 0, 0',
	X =  1662.442  mm,	Y = -1389.784  mm,	Z =  1034.707  mm,
	W =   -42.573 deg,	P =   -16.796 deg,	R =    43.536 deg
   GP2:
	UF : 1, UT : 1,
	J1=   180.000 deg,	J2=  -125.000 deg
};
P[747]{
   GP1:
	UF : 1, UT : 1,		CONFIG : 'N U T, 0, 0, 0',
	X =  1678.550  mm,	Y = -1382.945  mm,	Z =  1035.194  mm,
	W =   -43.824 deg,	P =   -18.067 deg,	R =    47.125 deg
   GP2:
	UF : 1, UT : 1,
	J1=   180.000 deg,	J2=  -125.000 deg
};
P[748]{
   GP1:
	UF : 1, UT : 1,		CONFIG : 'F U T, 0, 0, 0',
	X =  1100.081  mm,	Y =  1012.995  mm,	Z =  1030.748  mm,
	W =    44.134 deg,	P =    -6.199 deg,	R =   -51.547 deg
   GP2:
	UF : 1, UT : 1,
	J1=   180.000 deg,	J2=   150.000 deg
};
P[749]{
   GP1:
	UF : 1, UT : 1,		CONFIG : 'F U T, 0, 0, 0',
	X =  1113.832  mm,	Y =  1008.842  mm,	Z =  1030.040  mm,
	W =    43.018 deg,	P =    -7.263 deg,	R =   -34.945 deg
   GP2:
	UF : 1, UT : 1,
	J1=   180.000 deg,	J2=   150.000 deg
};
P[750]{
   GP1:
	UF : 1, UT : 1,		CONFIG : 'F U T, 0, 0, 0',
	X =  1124.302  mm,	Y =  1006.723  mm,	Z =  1029.912  mm,
	W =    42.651 deg,	P =   -14.125 deg,	R =   -20.717 deg
   GP2:
	UF : 1, UT : 1,
	J1=   180.000 deg,	J2=   150.000 deg
};
P[751]{
   GP1:
	UF : 1, UT : 1,		CONFIG : 'F U T, 0, 0, 0',
	X =  1138.783  mm,	Y =  1004.894  mm,	Z =  1031.267  mm,
	W =    42.647 deg,	P =   -14.130 deg,	R =   -27.081 deg
   GP2:
	UF : 1, UT : 1,
	J1=   180.000 deg,	J2=   150.000 deg
};
P[752]{
   GP1:
	UF : 1, UT : 1,		CONFIG : 'N U T, 0, 0, 0',
	X =  2793.017  mm,	Y = -1472.744  mm,	Z =   939.115  mm,
	W =   -37.776 deg,	P =   -31.389 deg,	R =    42.831 deg
   GP2:
	UF : 1, UT : 1,
	J1=   100.000 deg,	J2=   -90.000 deg
};
P[753]{
   GP1:
	UF : 1, UT : 1,		CONFIG : 'N U T, 0, 0, 0',
	X =  2794.995  mm,	Y = -1494.504  mm,	Z =   937.599  mm,
	W =   -37.762 deg,	P =   -31.393 deg,	R =    42.829 deg
   GP2:
	UF : 1, UT : 1,
	J1=   100.000 deg,	J2=   -90.000 deg
};
P[754]{
   GP1:
	UF : 1, UT : 1,		CONFIG : 'N U T, 0, 0, 0',
	X =  2786.501  mm,	Y = -1525.976  mm,	Z =   936.000  mm,
	W =   -42.869 deg,	P =   -22.972 deg,	R =    39.989 deg
   GP2:
	UF : 1, UT : 1,
	J1=    99.999 deg,	J2=   -90.000 deg
};
P[755]{
   GP1:
	UF : 1, UT : 1,		CONFIG : 'N U T, 0, 0, 0',
	X =  2776.812  mm,	Y = -1537.743  mm,	Z =   933.598  mm,
	W =   -45.701 deg,	P =   -14.897 deg,	R =    35.260 deg
   GP2:
	UF : 1, UT : 1,
	J1=   100.000 deg,	J2=   -90.000 deg
};
P[756]{
   GP1:
	UF : 1, UT : 1,		CONFIG : 'N U T, 0, 0, -1',
	X =  2500.465  mm,	Y = -1499.903  mm,	Z =  1059.350  mm,
	W =   -50.284 deg,	P =   -30.325 deg,	R =    67.097 deg
   GP2:
	UF : 0, UT : 1,
	J1=   100.000 deg,	J2=   -90.000 deg
};
P[757]{
   GP1:
	UF : 1, UT : 1,		CONFIG : 'N U T, 0, 0, 0',
	X =  2742.053  mm,	Y = -1559.698  mm,	Z =   926.134  mm,
	W =   -45.722 deg,	P =   -14.879 deg,	R =    30.415 deg
   GP2:
	UF : 1, UT : 1,
	J1=   100.000 deg,	J2=   -90.000 deg
};
P[758]{
   GP1:
	UF : 1, UT : 1,		CONFIG : 'N U T, 0, 0, 0',
	X =  2723.925  mm,	Y = -1565.150  mm,	Z =   922.276  mm,
	W =   -45.707 deg,	P =   -14.888 deg,	R =    18.304 deg
   GP2:
	UF : 1, UT : 1,
	J1=   100.000 deg,	J2=   -90.000 deg
};
P[759]{
   GP1:
	UF : 1, UT : 1,		CONFIG : 'N U T, 0, 0, 0',
	X =  2711.316  mm,	Y = -1566.584  mm,	Z =   918.265  mm,
	W =   -45.711 deg,	P =   -14.879 deg,	R =     6.076 deg
   GP2:
	UF : 1, UT : 1,
	J1=   100.000 deg,	J2=   -90.000 deg
};
P[760]{
   GP1:
	UF : 1, UT : 1,		CONFIG : 'N U T, 0, 0, 0',
	X =  2683.065  mm,	Y = -1567.564  mm,	Z =   912.242  mm,
	W =   -45.718 deg,	P =   -14.888 deg,	R =     6.082 deg
   GP2:
	UF : 1, UT : 1,
	J1=   100.000 deg,	J2=   -90.000 deg
};
P[761]{
   GP1:
	UF : 1, UT : 1,		CONFIG : 'N U T, 0, 0, 0',
	X =  2831.444  mm,	Y =  1497.758  mm,	Z =   887.365  mm,
	W =     1.873 deg,	P =   -42.067 deg,	R =    -2.897 deg
   GP2:
	UF : 1, UT : 1,
	J1=    95.000 deg,	J2=    90.000 deg
};
P[762]{
   GP1:
	UF : 1, UT : 1,		CONFIG : 'N U T, 0, 0, 0',
	X =  2831.262  mm,	Y =  1525.855  mm,	Z =   886.478  mm,
	W =     1.854 deg,	P =   -42.068 deg,	R =    -2.887 deg
   GP2:
	UF : 1, UT : 1,
	J1=    95.000 deg,	J2=    90.000 deg
};
P[763]{
   GP1:
	UF : 1, UT : 1,		CONFIG : 'N U T, 0, 0, 0',
	X =  2827.716  mm,	Y =  1550.337  mm,	Z =   883.519  mm,
	W =    47.255 deg,	P =   -13.928 deg,	R =   -43.726 deg
   GP2:
	UF : 1, UT : 1,
	J1=    95.000 deg,	J2=    90.000 deg
};
P[764]{
   GP1:
	UF : 1, UT : 1,		CONFIG : 'N U T, 0, 0, 0',
	X =  2804.967  mm,	Y =  1574.325  mm,	Z =   883.334  mm,
	W =    47.466 deg,	P =    -2.509 deg,	R =   -28.092 deg
   GP2:
	UF : 1, UT : 1,
	J1=    95.000 deg,	J2=    90.000 deg
};
P[765]{
   GP1:
	UF : 1, UT : 1,		CONFIG : 'N U T, 0, 0, 0',
	X =  2612.111  mm,	Y = -1537.301  mm,	Z =  1175.202  mm,
	W =   -45.531 deg,	P =     6.252 deg,	R =    32.963 deg
   GP2:
	UF : 0, UT : 1,
	J1=   100.000 deg,	J2=   -90.000 deg
};
P[766]{
   GP1:
	UF : 1, UT : 1,		CONFIG : 'N U T, 0, 0, 0',
	X =  2773.183  mm,	Y =  1590.041  mm,	Z =   880.231  mm,
	W =    47.470 deg,	P =    -2.509 deg,	R =   -28.100 deg
   GP2:
	UF : 1, UT : 1,
	J1=    95.000 deg,	J2=    90.000 deg
};
P[767]{
   GP1:
	UF : 1, UT : 1,		CONFIG : 'N U T, 0, 0, 0',
	X =  2764.750  mm,	Y =  1592.676  mm,	Z =   879.887  mm,
	W =    46.963 deg,	P =     8.290 deg,	R =   -26.942 deg
   GP2:
	UF : 1, UT : 1,
	J1=    95.000 deg,	J2=    90.000 deg
};
P[768]{
   GP1:
	UF : 1, UT : 1,		CONFIG : 'N U T, 0, 0, 0',
	X =  2755.466  mm,	Y =  1595.589  mm,	Z =   878.719  mm,
	W =    47.288 deg,	P =    13.426 deg,	R =   -20.074 deg
   GP2:
	UF : 1, UT : 1,
	J1=    94.995 deg,	J2=    90.000 deg
};
P[769]{
   GP1:
	UF : 1, UT : 1,		CONFIG : 'N U T, 0, 0, 0',
	X =  2714.916  mm,	Y =  1594.651  mm,	Z =   876.252  mm,
	W =    46.306 deg,	P =    12.117 deg,	R =   -20.583 deg
   GP2:
	UF : 1, UT : 1,
	J1=    95.000 deg,	J2=    90.000 deg
};
P[770]{
   GP1:
	UF : 1, UT : 1,		CONFIG : 'N U T, 0, 0, 0',
	X =  2775.833  mm,	Y =    59.955  mm,	Z =  -590.785  mm,
	W =     -.292 deg,	P =    37.605 deg,	R =      .743 deg
   GP2:
	UF : 1, UT : 1,
	J1=    90.000 deg,	J2=     0.000 deg
};
P[771]{
   GP1:
	UF : 1, UT : 1,		CONFIG : 'N U T, 0, 0, 0',
	X =  2775.834  mm,	Y =   -36.401  mm,	Z =  -590.784  mm,
	W =     -.292 deg,	P =    37.605 deg,	R =      .743 deg
   GP2:
	UF : 1, UT : 1,
	J1=    90.000 deg,	J2=     0.000 deg
};
P[772]{
   GP1:
	UF : 1, UT : 1,		CONFIG : 'N U T, 0, 0, 0',
	X =  2749.821  mm,	Y =   428.939  mm,	Z =   464.667  mm,
	W =    44.528 deg,	P =    -7.216 deg,	R =     7.296 deg
   GP2:
	UF : 1, UT : 1,
	J1=    90.000 deg,	J2=     0.000 deg
};
P[773]{
   GP1:
	UF : 1, UT : 1,		CONFIG : 'N U T, 0, 0, 0',
	X =  2715.354  mm,	Y =   428.138  mm,	Z =   464.592  mm,
	W =    44.543 deg,	P =    -7.213 deg,	R =     7.268 deg
   GP2:
	UF : 1, UT : 1,
	J1=    90.000 deg,	J2=     0.000 deg
};
P[774]{
   GP1:
	UF : 1, UT : 1,		CONFIG : 'N U T, 0, 0, 0',
	X =  2752.117  mm,	Y =  -403.442  mm,	Z =   463.818  mm,
	W =   -44.526 deg,	P =     7.212 deg,	R =     7.276 deg
   GP2:
	UF : 1, UT : 1,
	J1=    90.000 deg,	J2=     0.000 deg
};
P[775]{
   GP1:
	UF : 1, UT : 1,		CONFIG : 'N U T, 0, 0, 0',
	X =  2715.282  mm,	Y =  -404.077  mm,	Z =   462.987  mm,
	W =   -44.523 deg,	P =     7.209 deg,	R =     7.270 deg
   GP2:
	UF : 1, UT : 1,
	J1=    90.000 deg,	J2=     0.000 deg
};
P[776]{
   GP1:
	UF : 1, UT : 1,		CONFIG : 'F U T, 0, 0, 0',
	X =  2905.759  mm,	Y =   297.489  mm,	Z =   466.526  mm,
	W =   -14.926 deg,	P =   -42.904 deg,	R =    33.356 deg
   GP2:
	UF : 1, UT : 1,
	J1=    90.000 deg,	J2=     0.000 deg
};
P[777]{
   GP1:
	UF : 1, UT : 1,		CONFIG : 'F U T, 0, 0, 0',
	X =  2904.895  mm,	Y =   379.659  mm,	Z =   467.464  mm,
	W =    -8.441 deg,	P =   -43.927 deg,	R =    33.763 deg
   GP2:
	UF : 1, UT : 1,
	J1=    90.000 deg,	J2=     0.000 deg
};
P[778]{
   GP1:
	UF : 1, UT : 1,		CONFIG : 'N U T, 0, 0, 0',
	X =  1291.874  mm,	Y =   905.815  mm,	Z =  2427.792  mm,
	W =    68.242 deg,	P =   -43.563 deg,	R =   -51.949 deg
   GP2:
	UF : 1, UT : 1,
	J1=    95.000 deg,	J2=    90.000 deg
};
P[779]{
   GP1:
	UF : 1, UT : 1,		CONFIG : 'F U T, 0, 0, 0',
	X =  2904.123  mm,	Y =   411.321  mm,	Z =   468.436  mm,
	W =    -2.983 deg,	P =   -44.252 deg,	R =    40.170 deg
   GP2:
	UF : 1, UT : 1,
	J1=    90.000 deg,	J2=     0.000 deg
};
P[780]{
   GP1:
	UF : 1, UT : 1,		CONFIG : 'N U T, 0, 0, 0',
	X =  2526.820  mm,	Y =  1556.392  mm,	Z =  1079.609  mm,
	W =    21.780 deg,	P =   -40.404 deg,	R =   -29.962 deg
   GP2:
	UF : 0, UT : 1,
	J1=    95.000 deg,	J2=    90.000 deg
};
P[781]{
   GP1:
	UF : 1, UT : 1,		CONFIG : 'N U T, 0, 0, 0',
	X =  2659.725  mm,	Y =  1505.803  mm,	Z =  1079.609  mm,
	W =    15.908 deg,	P =   -31.536 deg,	R =   -26.500 deg
   GP2:
	UF : 0, UT : 1,
	J1=    95.000 deg,	J2=    90.000 deg
};
P[782]{
   GP1:
	UF : 1, UT : 1,		CONFIG : 'F U T, 0, 0, 0',
	X =  2902.073  mm,	Y =   421.602  mm,	Z =   467.948  mm,
	W =    -2.617 deg,	P =   -43.939 deg,	R =    53.826 deg
   GP2:
	UF : 1, UT : 1,
	J1=    90.000 deg,	J2=     0.000 deg
};
P[783]{
   GP1:
	UF : 1, UT : 1,		CONFIG : 'F U T, 0, 0, 0',
	X =  2887.593  mm,	Y =   431.459  mm,	Z =   467.662  mm,
	W =    -2.617 deg,	P =   -43.939 deg,	R =    78.094 deg
   GP2:
	UF : 1, UT : 1,
	J1=    90.000 deg,	J2=     0.000 deg
};
P[784]{
   GP1:
	UF : 1, UT : 1,		CONFIG : 'F U T, 0, 0, 0',
	X =  2878.735  mm,	Y =   431.459  mm,	Z =   467.662  mm,
	W =    -2.617 deg,	P =   -43.939 deg,	R =    78.094 deg
   GP2:
	UF : 1, UT : 1,
	J1=    90.000 deg,	J2=     0.000 deg
};
P[785]{
   GP1:
	UF : 1, UT : 1,		CONFIG : 'N U T, 0, 0, 0',
	X =  2903.526  mm,	Y =  -269.076  mm,	Z =   466.198  mm,
	W =    14.881 deg,	P =   -42.512 deg,	R =   -27.203 deg
   GP2:
	UF : 1, UT : 1,
	J1=    90.000 deg,	J2=     0.000 deg
};
P[786]{
   GP1:
	UF : 1, UT : 1,		CONFIG : 'N U T, 0, 0, 0',
	X =  2902.858  mm,	Y =  -366.735  mm,	Z =   467.050  mm,
	W =     7.402 deg,	P =   -43.864 deg,	R =   -27.796 deg
   GP2:
	UF : 1, UT : 1,
	J1=    90.000 deg,	J2=     0.000 deg
};
P[787]{
   GP1:
	UF : 1, UT : 1,		CONFIG : 'N U T, 0, 0, 0',
	X =  2902.317  mm,	Y =  -381.646  mm,	Z =   467.885  mm,
	W =     7.404 deg,	P =   -43.863 deg,	R =   -33.013 deg
   GP2:
	UF : 1, UT : 1,
	J1=    90.000 deg,	J2=     0.000 deg
};
P[788]{
   GP1:
	UF : 1, UT : 1,		CONFIG : 'N U T, 0, 0, 0',
	X =  2895.908  mm,	Y =  -394.691  mm,	Z =   467.867  mm,
	W =    -1.094 deg,	P =   -44.445 deg,	R =   -50.602 deg
   GP2:
	UF : 1, UT : 1,
	J1=    89.996 deg,	J2=     0.000 deg
};
P[789]{
   GP1:
	UF : 1, UT : 1,		CONFIG : 'N U T, 0, 0, 0',
	X =  2889.336  mm,	Y =  -400.456  mm,	Z =   464.138  mm,
	W =    -1.103 deg,	P =   -44.447 deg,	R =   -71.047 deg
   GP2:
	UF : 1, UT : 1,
	J1=    89.995 deg,	J2=     0.000 deg
};
P[790]{
   GP1:
	UF : 1, UT : 1,		CONFIG : 'N U T, 0, 0, 0',
	X =  2586.641  mm,	Y =  1526.023  mm,	Z =  1082.786  mm,
	W =    42.689 deg,	P =    16.599 deg,	R =   -42.374 deg
   GP2:
	UF : 0, UT : 1,
	J1=    95.000 deg,	J2=    90.000 deg
};
P[791]{
   GP1:
	UF : 1, UT : 1,		CONFIG : 'N U T, 0, 0, 0',
	X =  2877.924  mm,	Y =  -402.031  mm,	Z =   463.256  mm,
	W =    -1.100 deg,	P =   -44.451 deg,	R =   -71.051 deg
   GP2:
	UF : 1, UT : 1,
	J1=    89.995 deg,	J2=     0.000 deg
};
P[792]{
   GP1:
	UF : 1, UT : 1,		CONFIG : 'F U T, 0, 0, 0',
	X =  2905.759  mm,	Y =   297.489  mm,	Z =   466.526  mm,
	W =   -14.926 deg,	P =   -42.904 deg,	R =    33.356 deg
   GP2:
	UF : 1, UT : 1,
	J1=    90.000 deg,	J2=     0.000 deg
};
P[793]{
   GP1:
	UF : 1, UT : 1,		CONFIG : 'F U T, 0, 0, 0',
	X =   419.331  mm,	Y =  1026.789  mm,	Z =  1609.020  mm,
	W =    71.318 deg,	P =     7.769 deg,	R =   -20.454 deg
   GP2:
	UF : 1, UT : 1,
	J1=   180.000 deg,	J2=   150.000 deg
};
P[794]{
   GP1:
	UF : 1, UT : 1,		CONFIG : 'F U T, 0, 0, 0',
	X =  2904.895  mm,	Y =   379.659  mm,	Z =   467.464  mm,
	W =    -8.441 deg,	P =   -43.927 deg,	R =    33.763 deg
   GP2:
	UF : 1, UT : 1,
	J1=    90.000 deg,	J2=     0.000 deg
};
P[795]{
   GP1:
	UF : 1, UT : 1,		CONFIG : 'F U T, 0, 0, 0',
	X =  2904.123  mm,	Y =   411.321  mm,	Z =   468.436  mm,
	W =    -2.983 deg,	P =   -44.252 deg,	R =    40.170 deg
   GP2:
	UF : 1, UT : 1,
	J1=    90.000 deg,	J2=     0.000 deg
};
P[796]{
   GP1:
	UF : 1, UT : 1,		CONFIG : 'F U T, 0, 0, 0',
	X =  2902.073  mm,	Y =   421.602  mm,	Z =   467.948  mm,
	W =    -2.617 deg,	P =   -43.939 deg,	R =    53.826 deg
   GP2:
	UF : 1, UT : 1,
	J1=    90.000 deg,	J2=     0.000 deg
};
P[797]{
   GP1:
	UF : 1, UT : 1,		CONFIG : 'F U T, 0, 0, 0',
	X =  2887.593  mm,	Y =   431.459  mm,	Z =   467.662  mm,
	W =    -2.617 deg,	P =   -43.939 deg,	R =    78.094 deg
   GP2:
	UF : 1, UT : 1,
	J1=    90.000 deg,	J2=     0.000 deg
};
P[798]{
   GP1:
	UF : 1, UT : 1,		CONFIG : 'F U T, 0, 0, 0',
	X =  2878.735  mm,	Y =   431.459  mm,	Z =   467.662  mm,
	W =    -2.617 deg,	P =   -43.939 deg,	R =    78.094 deg
   GP2:
	UF : 1, UT : 1,
	J1=    90.000 deg,	J2=     0.000 deg
};
P[799]{
   GP1:
	UF : 1, UT : 1,		CONFIG : 'F U T, 0, 0, 0',
	X =  2905.759  mm,	Y =   297.489  mm,	Z =   466.526  mm,
	W =   -14.926 deg,	P =   -42.904 deg,	R =    33.356 deg
   GP2:
	UF : 1, UT : 1,
	J1=    90.000 deg,	J2=     0.000 deg
};
P[800]{
   GP1:
	UF : 1, UT : 1,		CONFIG : 'F U T, 0, 0, 0',
	X =  2904.895  mm,	Y =   379.659  mm,	Z =   467.464  mm,
	W =    -8.441 deg,	P =   -43.927 deg,	R =    33.763 deg
   GP2:
	UF : 1, UT : 1,
	J1=    90.000 deg,	J2=     0.000 deg
};
P[801]{
   GP1:
	UF : 1, UT : 1,		CONFIG : 'F U T, 0, 0, 0',
	X =  2904.123  mm,	Y =   411.321  mm,	Z =   468.436  mm,
	W =    -2.983 deg,	P =   -44.252 deg,	R =    40.170 deg
   GP2:
	UF : 1, UT : 1,
	J1=    90.000 deg,	J2=     0.000 deg
};
P[802]{
   GP1:
	UF : 1, UT : 1,		CONFIG : 'F U T, 0, 0, 0',
	X =  2902.073  mm,	Y =   421.602  mm,	Z =   467.948  mm,
	W =    -2.617 deg,	P =   -43.939 deg,	R =    53.826 deg
   GP2:
	UF : 1, UT : 1,
	J1=    90.000 deg,	J2=     0.000 deg
};
P[803]{
   GP1:
	UF : 1, UT : 1,		CONFIG : 'F U T, 0, 0, 0',
	X =  2887.593  mm,	Y =   431.459  mm,	Z =   467.662  mm,
	W =    -2.617 deg,	P =   -43.939 deg,	R =    78.094 deg
   GP2:
	UF : 1, UT : 1,
	J1=    90.000 deg,	J2=     0.000 deg
};
P[804]{
   GP1:
	UF : 1, UT : 1,		CONFIG : 'F U T, 0, 0, 0',
	X =  2878.735  mm,	Y =   431.459  mm,	Z =   467.662  mm,
	W =    -2.617 deg,	P =   -43.939 deg,	R =    78.094 deg
   GP2:
	UF : 1, UT : 1,
	J1=    90.000 deg,	J2=     0.000 deg
};
P[805]{
   GP1:
	UF : 1, UT : 1,		CONFIG : 'N U T, 0, 0, 0',
	X =  2903.526  mm,	Y =  -269.076  mm,	Z =   466.198  mm,
	W =    14.881 deg,	P =   -42.512 deg,	R =   -27.203 deg
   GP2:
	UF : 1, UT : 1,
	J1=    90.000 deg,	J2=     0.000 deg
};
P[806]{
   GP1:
	UF : 1, UT : 1,		CONFIG : 'N U T, 0, 0, 0',
	X =  2902.858  mm,	Y =  -366.735  mm,	Z =   467.050  mm,
	W =     7.402 deg,	P =   -43.864 deg,	R =   -27.796 deg
   GP2:
	UF : 1, UT : 1,
	J1=    90.000 deg,	J2=     0.000 deg
};
P[807]{
   GP1:
	UF : 1, UT : 1,		CONFIG : 'N U T, 0, 0, 0',
	X =  2902.317  mm,	Y =  -381.646  mm,	Z =   467.885  mm,
	W =     7.404 deg,	P =   -43.863 deg,	R =   -33.013 deg
   GP2:
	UF : 1, UT : 1,
	J1=    90.000 deg,	J2=     0.000 deg
};
P[808]{
   GP1:
	UF : 1, UT : 1,		CONFIG : 'N U T, 0, 0, 0',
	X =  2895.908  mm,	Y =  -394.691  mm,	Z =   467.867  mm,
	W =    -1.094 deg,	P =   -44.445 deg,	R =   -50.602 deg
   GP2:
	UF : 1, UT : 1,
	J1=    89.996 deg,	J2=     0.000 deg
};
P[809]{
   GP1:
	UF : 1, UT : 1,		CONFIG : 'N U T, 0, 0, 0',
	X =  2889.336  mm,	Y =  -400.456  mm,	Z =   464.138  mm,
	W =    -1.103 deg,	P =   -44.447 deg,	R =   -71.047 deg
   GP2:
	UF : 1, UT : 1,
	J1=    89.995 deg,	J2=     0.000 deg
};
P[810]{
   GP1:
	UF : 1, UT : 1,		CONFIG : 'N U T, 0, 0, 0',
	X =  2877.924  mm,	Y =  -402.031  mm,	Z =   463.256  mm,
	W =    -1.100 deg,	P =   -44.451 deg,	R =   -71.051 deg
   GP2:
	UF : 1, UT : 1,
	J1=    89.995 deg,	J2=     0.000 deg
};
P[811]{
   GP1:
	UF : 1, UT : 1,		CONFIG : 'N U T, 0, 0, 0',
	X =  2903.526  mm,	Y =  -269.076  mm,	Z =   466.198  mm,
	W =    14.881 deg,	P =   -42.512 deg,	R =   -27.203 deg
   GP2:
	UF : 1, UT : 1,
	J1=    90.000 deg,	J2=     0.000 deg
};
P[812]{
   GP1:
	UF : 1, UT : 1,		CONFIG : 'N U T, 0, 0, 0',
	X =  2902.858  mm,	Y =  -366.735  mm,	Z =   467.050  mm,
	W =     7.402 deg,	P =   -43.864 deg,	R =   -27.796 deg
   GP2:
	UF : 1, UT : 1,
	J1=    90.000 deg,	J2=     0.000 deg
};
P[813]{
   GP1:
	UF : 1, UT : 1,		CONFIG : 'N U T, 0, 0, 0',
	X =  2902.317  mm,	Y =  -381.646  mm,	Z =   467.885  mm,
	W =     7.404 deg,	P =   -43.863 deg,	R =   -33.013 deg
   GP2:
	UF : 1, UT : 1,
	J1=    90.000 deg,	J2=     0.000 deg
};
P[814]{
   GP1:
	UF : 1, UT : 1,		CONFIG : 'N U T, 0, 0, 0',
	X =  2895.908  mm,	Y =  -394.691  mm,	Z =   467.867  mm,
	W =    -1.094 deg,	P =   -44.445 deg,	R =   -50.602 deg
   GP2:
	UF : 1, UT : 1,
	J1=    89.996 deg,	J2=     0.000 deg
};
P[815]{
   GP1:
	UF : 1, UT : 1,		CONFIG : 'N U T, 0, 0, 0',
	X =  2889.336  mm,	Y =  -400.456  mm,	Z =   464.138  mm,
	W =    -1.103 deg,	P =   -44.447 deg,	R =   -71.047 deg
   GP2:
	UF : 1, UT : 1,
	J1=    89.995 deg,	J2=     0.000 deg
};
P[816]{
   GP1:
	UF : 1, UT : 1,		CONFIG : 'N U T, 0, 0, 0',
	X =  2877.924  mm,	Y =  -402.031  mm,	Z =   463.256  mm,
	W =    -1.100 deg,	P =   -44.451 deg,	R =   -71.051 deg
   GP2:
	UF : 1, UT : 1,
	J1=    89.995 deg,	J2=     0.000 deg
};
P[817]{
   GP1:
	UF : 1, UT : 1,		CONFIG : 'N U T, 0, 0, 1',
	X =  2745.545  mm,	Y =  -276.052  mm,	Z =   464.654  mm,
	W =    29.147 deg,	P =    30.453 deg,	R =  -132.266 deg
   GP2:
	UF : 1, UT : 1,
	J1=    90.000 deg,	J2=     0.000 deg
};
P[818]{
   GP1:
	UF : 1, UT : 1,		CONFIG : 'N U T, 0, 0, 1',
	X =  2745.001  mm,	Y =  -318.060  mm,	Z =   465.700  mm,
	W =    29.459 deg,	P =    30.698 deg,	R =  -132.107 deg
   GP2:
	UF : 1, UT : 1,
	J1=    90.000 deg,	J2=     0.000 deg
};
P[819]{
   GP1:
	UF : 1, UT : 1,		CONFIG : 'N U T, 0, 0, 1',
	X =  2759.258  mm,	Y =  -343.755  mm,	Z =   464.873  mm,
	W =    32.708 deg,	P =    26.756 deg,	R =  -103.211 deg
   GP2:
	UF : 1, UT : 1,
	J1=    90.000 deg,	J2=     0.000 deg
};
P[820]{
   GP1:
	UF : 1, UT : 1,		CONFIG : 'N U T, 0, 0, 0',
	X =  2781.851  mm,	Y =  -350.503  mm,	Z =   466.805  mm,
	W =    32.871 deg,	P =    19.630 deg,	R =   -83.146 deg
   GP2:
	UF : 1, UT : 1,
	J1=    90.000 deg,	J2=     0.000 deg
};
P[821]{
   GP1:
	UF : 1, UT : 1,		CONFIG : 'N U T, 0, 0, 0',
	X =  2740.523  mm,	Y =   300.010  mm,	Z =   465.528  mm,
	W =   -36.614 deg,	P =    28.247 deg,	R =   122.490 deg
   GP2:
	UF : 1, UT : 1,
	J1=    90.000 deg,	J2=     0.000 deg
};
P[822]{
   GP1:
	UF : 1, UT : 1,		CONFIG : 'N U T, 0, 0, 0',
	X =  2741.022  mm,	Y =   348.224  mm,	Z =   465.529  mm,
	W =   -36.614 deg,	P =    28.247 deg,	R =   122.490 deg
   GP2:
	UF : 1, UT : 1,
	J1=    90.000 deg,	J2=     0.000 deg
};
P[823]{
   GP1:
	UF : 1, UT : 1,		CONFIG : 'N U T, 0, 0, 0',
	X =  2758.912  mm,	Y =   371.174  mm,	Z =   466.650  mm,
	W =   -32.204 deg,	P =    27.169 deg,	R =   100.051 deg
   GP2:
	UF : 1, UT : 1,
	J1=    90.000 deg,	J2=     0.000 deg
};
P[824]{
   GP1:
	UF : 1, UT : 1,		CONFIG : 'N U T, 0, 0, 0',
	X =  2774.997  mm,	Y =   375.066  mm,	Z =   468.013  mm,
	W =   -28.646 deg,	P =    22.121 deg,	R =    94.724 deg
   GP2:
	UF : 1, UT : 1,
	J1=    90.000 deg,	J2=     0.000 deg
};
P[825]{
   GP1:
	UF : 1, UT : 1,		CONFIG : 'N U T, 0, 0, 0',
	X =  1668.877  mm,	Y =   251.121  mm,	Z =   363.698  mm,
	W =    31.331 deg,	P =    33.498 deg,	R =    49.952 deg
   GP2:
	UF : 1, UT : 1,
	J1=    90.000 deg,	J2=     0.000 deg
};
P[826]{
   GP1:
	UF : 1, UT : 1,		CONFIG : 'N U T, 0, 0, 0',
	X =  1668.020  mm,	Y =   178.121  mm,	Z =   363.698  mm,
	W =    31.331 deg,	P =    33.498 deg,	R =    49.952 deg
   GP2:
	UF : 1, UT : 1,
	J1=    90.000 deg,	J2=     0.000 deg
};
P[827]{
   GP1:
	UF : 1, UT : 1,		CONFIG : 'N U T, 0, 0, 0',
	X =  1671.284  mm,	Y =  -228.674  mm,	Z =   362.649  mm,
	W =   -34.074 deg,	P =    31.387 deg,	R =   -56.109 deg
   GP2:
	UF : 1, UT : 1,
	J1=    90.000 deg,	J2=     0.000 deg
};
P[828]{
   GP1:
	UF : 1, UT : 1,		CONFIG : 'N U T, 0, 0, 0',
	X =  1671.070  mm,	Y =  -158.103  mm,	Z =   362.293  mm,
	W =   -34.074 deg,	P =    31.387 deg,	R =   -56.109 deg
   GP2:
	UF : 1, UT : 1,
	J1=    90.000 deg,	J2=     0.000 deg
};
P[829]{
   GP1:
	UF : 1, UT : 1,		CONFIG : 'N U T, 0, 0, 0',
	X =  1808.570  mm,	Y =  -390.427  mm,	Z =   832.270  mm,
	W =     -.610 deg,	P =      .928 deg,	R =   -33.342 deg
   GP2:
	UF : 1, UT : 1,
	J1=    45.000 deg,	J2=     0.000 deg
};
P[830]{
   GP1:
	UF : 1, UT : 1,		CONFIG : 'N U T, 0, 0, 0',
	X =  1807.828  mm,	Y =  -159.968  mm,	Z =   830.736  mm,
	W =     -.607 deg,	P =      .924 deg,	R =   -33.344 deg
   GP2:
	UF : 1, UT : 1,
	J1=    45.000 deg,	J2=     0.000 deg
};
P[831]{
   GP1:
	UF : 1, UT : 1,		CONFIG : 'N U T, 0, 0, 0',
	X =  1804.560  mm,	Y =   408.326  mm,	Z =   829.592  mm,
	W =     -.607 deg,	P =      .924 deg,	R =    40.442 deg
   GP2:
	UF : 1, UT : 1,
	J1=    45.000 deg,	J2=     0.000 deg
};
P[832]{
   GP1:
	UF : 1, UT : 1,		CONFIG : 'N U T, 0, 0, 0',
	X =  1806.042  mm,	Y =   179.612  mm,	Z =   828.163  mm,
	W =     -.607 deg,	P =      .924 deg,	R =    40.442 deg
   GP2:
	UF : 1, UT : 1,
	J1=    45.000 deg,	J2=     0.000 deg
};
P[833]{
   GP1:
	UF : 1, UT : 1,		CONFIG : 'N U T, 0, 0, 0',
	X =  2178.657  mm,	Y =   659.349  mm,	Z =  1322.478  mm,
	W =     -.151 deg,	P =     4.190 deg,	R =     -.119 deg
   GP2:
	UF : 1, UT : 1,
	J1=   124.996 deg,	J2=     0.000 deg
};
P[834]{
   GP1:
	UF : 1, UT : 1,		CONFIG : 'N U T, 0, 0, 0',
	X =  2179.570  mm,	Y =   501.982  mm,	Z =  1322.098  mm,
	W =      .050 deg,	P =     4.374 deg,	R =     -.049 deg
   GP2:
	UF : 1, UT : 1,
	J1=   124.995 deg,	J2=     0.000 deg
};
P[835]{
   GP1:
	UF : 1, UT : 1,		CONFIG : 'N U T, 0, 0, 0',
	X =  2179.470  mm,	Y =   459.845  mm,	Z =  1322.928  mm,
	W =   -10.985 deg,	P =     4.746 deg,	R =     -.446 deg
   GP2:
	UF : 1, UT : 1,
	J1=   124.999 deg,	J2=     0.000 deg
};
P[836]{
   GP1:
	UF : 1, UT : 1,		CONFIG : 'N U T, 0, 0, 0',
	X =  2167.431  mm,	Y =    27.132  mm,	Z =  1339.879  mm,
	W =     -.713 deg,	P =     8.623 deg,	R =     -.119 deg
   GP2:
	UF : 1, UT : 1,
	J1=   124.996 deg,	J2=     0.000 deg
};
P[837]{
   GP1:
	UF : 1, UT : 1,		CONFIG : 'N U T, 0, 0, 0',
	X =  2168.446  mm,	Y =  -166.967  mm,	Z =  1339.463  mm,
	W =     -.016 deg,	P =    10.106 deg,	R =      .980 deg
   GP2:
	UF : 1, UT : 1,
	J1=   125.000 deg,	J2=     0.000 deg
};
P[838]{
   GP1:
	UF : 1, UT : 1,		CONFIG : 'N U T, 0, 0, 0',
	X =  2169.557  mm,	Y =  -389.532  mm,	Z =  1339.244  mm,
	W =     -.928 deg,	P =     7.504 deg,	R =     -.096 deg
   GP2:
	UF : 1, UT : 1,
	J1=   125.000 deg,	J2=     0.000 deg
};
P[839]{
   GP1:
	UF : 1, UT : 1,		CONFIG : 'N U T, 0, 0, 0',
	X =  2165.947  mm,	Y =   412.114  mm,	Z =  1341.826  mm,
	W =      .150 deg,	P =     6.214 deg,	R =      .016 deg
   GP2:
	UF : 1, UT : 1,
	J1=   125.000 deg,	J2=     0.000 deg
};
P[840]{
   GP1:
	UF : 1, UT : 1,		CONFIG : 'N U T, 0, 0, 0',
	X =  2167.028  mm,	Y =   193.246  mm,	Z =  1340.156  mm,
	W =      .990 deg,	P =     7.423 deg,	R =      .117 deg
   GP2:
	UF : 1, UT : 1,
	J1=   125.000 deg,	J2=     0.000 deg
};
P[841]{
   GP1:
	UF : 1, UT : 1,		CONFIG : 'N U T, 0, 0, 0',
	X =  2168.042  mm,	Y =    21.221  mm,	Z =  1339.306  mm,
	W =    -1.723 deg,	P =     8.124 deg,	R =     2.334 deg
   GP2:
	UF : 1, UT : 1,
	J1=   125.000 deg,	J2=     0.000 deg
};
P[842]{
   GP1:
	UF : 1, UT : 1,		CONFIG : 'N U T, 0, 0, 0',
	X =  2183.748  mm,	Y =  -629.768  mm,	Z =  1321.915  mm,
	W =      .004 deg,	P =     8.094 deg,	R =      .009 deg
   GP2:
	UF : 1, UT : 1,
	J1=   125.000 deg,	J2=     0.000 deg
};
P[843]{
   GP1:
	UF : 1, UT : 1,		CONFIG : 'N U T, 0, 0, 0',
	X =  2183.088  mm,	Y =  -436.975  mm,	Z =  1322.259  mm,
	W =      .023 deg,	P =     7.896 deg,	R =     -.019 deg
   GP2:
	UF : 1, UT : 1,
	J1=   125.000 deg,	J2=     0.000 deg
};
P[844]{
   GP1:
	UF : 1, UT : 1,		CONFIG : 'N U T, 0, 0, 0',
	X =  2182.831  mm,	Y =  -431.800  mm,	Z =  1321.998  mm,
	W =     8.588 deg,	P =     5.688 deg,	R =      .847 deg
   GP2:
	UF : 1, UT : 1,
	J1=   125.000 deg,	J2=     0.000 deg
};
P[845]{
   GP1:
	UF : 1, UT : 1,		CONFIG : 'N U T, 0, 0, 0',
	X =  2136.258  mm,	Y =   423.750  mm,	Z =   282.790  mm,
	W =    39.277 deg,	P =    23.849 deg,	R =     9.150 deg
   GP2:
	UF : 1, UT : 1,
	J1=     0.000 deg,	J2=   180.000 deg
};
P[846]{
   GP1:
	UF : 1, UT : 1,		CONFIG : 'N U T, 0, 0, 0',
	X =  2155.097  mm,	Y =   424.295  mm,	Z =   280.001  mm,
	W =    39.267 deg,	P =    23.856 deg,	R =   -24.748 deg
   GP2:
	UF : 1, UT : 1,
	J1=     0.000 deg,	J2=   180.000 deg
};
P[847]{
   GP1:
	UF : 1, UT : 1,		CONFIG : 'N U T, 0, 0, 0',
	X =  2191.038  mm,	Y =   425.038  mm,	Z =   280.145  mm,
	W =    39.348 deg,	P =    23.574 deg,	R =   -24.954 deg
   GP2:
	UF : 1, UT : 1,
	J1=     0.000 deg,	J2=   180.000 deg
};
P[848]{
   GP1:
	UF : 1, UT : 1,		CONFIG : 'N U T, 0, 0, 0',
	X =  2201.796  mm,	Y =   419.697  mm,	Z =   288.204  mm,
	W =    48.341 deg,	P =     9.057 deg,	R =   -36.927 deg
   GP2:
	UF : 1, UT : 1,
	J1=     0.000 deg,	J2=   180.000 deg
};
P[849]{
   GP1:
	UF : 1, UT : 1,		CONFIG : 'N U T, 0, 0, 0',
	X =  2125.458  mm,	Y =  -402.882  mm,	Z =   276.210  mm,
	W =   -42.888 deg,	P =    -2.088 deg,	R =   -37.991 deg
   GP2:
	UF : 1, UT : 1,
	J1=     0.000 deg,	J2=   180.000 deg
};
P[850]{
   GP1:
	UF : 1, UT : 1,		CONFIG : 'N U T, 0, 0, 0',
	X =  2146.996  mm,	Y =  -401.034  mm,	Z =   278.267  mm,
	W =   -42.902 deg,	P =    -2.083 deg,	R =    -3.515 deg
   GP2:
	UF : 1, UT : 1,
	J1=     0.000 deg,	J2=   180.000 deg
};
P[851]{
   GP1:
	UF : 1, UT : 1,		CONFIG : 'N U T, 0, 0, 0',
	X =  2201.068  mm,	Y =  -403.642  mm,	Z =   276.795  mm,
	W =   -42.889 deg,	P =    -2.090 deg,	R =    -3.521 deg
   GP2:
	UF : 1, UT : 1,
	J1=     0.000 deg,	J2=   180.000 deg
};
P[852]{
   GP1:
	UF : 1, UT : 1,		CONFIG : 'N U T, 0, 0, 0',
	X =  2208.911  mm,	Y =  -404.418  mm,	Z =   278.857  mm,
	W =   -37.665 deg,	P =   -22.310 deg,	R =     8.929 deg
   GP2:
	UF : 1, UT : 1,
	J1=     0.000 deg,	J2=   180.000 deg
};
P[853]{
   GP1:
	UF : 1, UT : 1,		CONFIG : 'N U T, 0, 0, 1',
	X =  2235.739  mm,	Y =  -233.047  mm,	Z =  -188.744  mm,
	W =    34.819 deg,	P =    27.070 deg,	R =  -123.447 deg
   GP2:
	UF : 1, UT : 1,
	J1=     0.000 deg,	J2=   180.000 deg
};
P[854]{
   GP1:
	UF : 1, UT : 1,		CONFIG : 'N U T, 0, 0, 1',
	X =  2233.830  mm,	Y =    -8.684  mm,	Z =  -186.712  mm,
	W =    34.826 deg,	P =    27.081 deg,	R =  -123.458 deg
   GP2:
	UF : 1, UT : 1,
	J1=     0.000 deg,	J2=   180.000 deg
};
P[855]{
   GP1:
	UF : 1, UT : 1,		CONFIG : 'N U T, 0, 0, 1',
	X =  2234.912  mm,	Y =    11.625  mm,	Z =  -185.523  mm,
	W =    33.015 deg,	P =    26.717 deg,	R =   -93.423 deg
   GP2:
	UF : 1, UT : 1,
	J1=     0.000 deg,	J2=   180.000 deg
};
P[856]{
   GP1:
	UF : 1, UT : 1,		CONFIG : 'N U T, 0, 0, 0',
	X =  2233.192  mm,	Y =   249.052  mm,	Z =  -187.235  mm,
	W =   -26.756 deg,	P =    37.337 deg,	R =   139.556 deg
   GP2:
	UF : 1, UT : 1,
	J1=     0.000 deg,	J2=   180.000 deg
};
P[857]{
   GP1:
	UF : 1, UT : 1,		CONFIG : 'N U T, 0, 0, 0',
	X =  2237.745  mm,	Y =    33.563  mm,	Z =  -188.748  mm,
	W =   -26.755 deg,	P =    37.337 deg,	R =   139.561 deg
   GP2:
	UF : 1, UT : 1,
	J1=     0.000 deg,	J2=   180.000 deg
};
P[858]{
   GP1:
	UF : 1, UT : 1,		CONFIG : 'N U T, 0, 0, 0',
	X =  2232.730  mm,	Y =     3.648  mm,	Z =  -186.256  mm,
	W =   -20.117 deg,	P =    35.519 deg,	R =   111.507 deg
   GP2:
	UF : 1, UT : 1,
	J1=     0.000 deg,	J2=   180.000 deg
};
P[859]{
   GP1:
	UF : 1, UT : 1,		CONFIG : 'N U T, 0, 0, 1',
	X =  1487.823  mm,	Y =  -637.223  mm,	Z =     4.887  mm,
	W =    42.306 deg,	P =    16.820 deg,	R =  -100.933 deg
   GP2:
	UF : 1, UT : 1,
	J1=     0.000 deg,	J2=   180.000 deg
};
P[860]{
   GP1:
	UF : 1, UT : 1,		CONFIG : 'N U T, 0, 0, 1',
	X =  1488.724  mm,	Y =  -603.338  mm,	Z =     5.170  mm,
	W =    42.315 deg,	P =    16.837 deg,	R =  -100.936 deg
   GP2:
	UF : 1, UT : 1,
	J1=     0.000 deg,	J2=   180.000 deg
};
P[861]{
   GP1:
	UF : 1, UT : 1,		CONFIG : 'N U T, 0, 0, 1',
	X =  1485.624  mm,	Y =  -440.808  mm,	Z =     7.456  mm,
	W =    42.350 deg,	P =    16.907 deg,	R =   -86.948 deg
   GP2:
	UF : 1, UT : 1,
	J1=     0.000 deg,	J2=   180.000 deg
};
P[862]{
   GP1:
	UF : 1, UT : 1,		CONFIG : 'N U T, 0, 0, 0',
	X =  1462.579  mm,	Y =    13.411  mm,	Z =     4.510  mm,
	W =      .947 deg,	P =    42.922 deg,	R =   177.955 deg
   GP2:
	UF : 1, UT : 1,
	J1=     0.000 deg,	J2=   180.000 deg
};
P[863]{
   GP1:
	UF : 1, UT : 1,		CONFIG : 'N U T, 0, 0, 1',
	X =  1463.463  mm,	Y =  -315.428  mm,	Z =     5.740  mm,
	W =    -1.380 deg,	P =    43.931 deg,	R =   175.837 deg
   GP2:
	UF : 1, UT : 1,
	J1=     0.000 deg,	J2=   180.000 deg
};
P[864]{
   GP1:
	UF : 1, UT : 1,		CONFIG : 'N U T, 0, 0, 1',
	X =  1462.309  mm,	Y =  -379.397  mm,	Z =     6.892  mm,
	W =     5.165 deg,	P =    43.293 deg,	R =  -179.580 deg
   GP2:
	UF : 1, UT : 1,
	J1=     0.000 deg,	J2=   180.000 deg
};
P[865]{
   GP1:
	UF : 1, UT : 1,		CONFIG : 'N U T, 0, 0, 0',
	X =  1459.882  mm,	Y =   397.906  mm,	Z =     4.916  mm,
	W =   -18.718 deg,	P =    37.733 deg,	R =   149.446 deg
   GP2:
	UF : 1, UT : 1,
	J1=     0.000 deg,	J2=   180.000 deg
};
P[866]{
   GP1:
	UF : 1, UT : 1,		CONFIG : 'N U T, 0, 0, 0',
	X =  1458.720  mm,	Y =    13.774  mm,	Z =     7.353  mm,
	W =      .274 deg,	P =    41.497 deg,	R =   174.619 deg
   GP2:
	UF : 1, UT : 1,
	J1=     0.000 deg,	J2=   180.000 deg
};
P[867]{
   GP1:
	UF : 1, UT : 1,		CONFIG : 'N U T, 0, 0, -1',
	X =  1483.448  mm,	Y =   656.175  mm,	Z =    14.251  mm,
	W =    29.504 deg,	P =    31.493 deg,	R =  -136.893 deg
   GP2:
	UF : 1, UT : 1,
	J1=     0.000 deg,	J2=   180.000 deg
};
P[868]{
   GP1:
	UF : 1, UT : 1,		CONFIG : 'N U T, 0, 0, -1',
	X =  1482.620  mm,	Y =   468.746  mm,	Z =    12.817  mm,
	W =    40.718 deg,	P =    18.744 deg,	R =  -126.943 deg
   GP2:
	UF : 1, UT : 1,
	J1=     0.000 deg,	J2=   180.000 deg
};
P[869]{
   GP1:
	UF : 1, UT : 1,		CONFIG : 'N U T, 0, 0, -1',
	X =  1482.535  mm,	Y =   458.132  mm,	Z =    12.780  mm,
	W =    41.200 deg,	P =    17.928 deg,	R =  -126.514 deg
   GP2:
	UF : 1, UT : 1,
	J1=     0.000 deg,	J2=   180.000 deg
};
P[870]{
   GP1:
	UF : 1, UT : 1,		CONFIG : 'N U T, 0, 0, 0',
	X =  2192.201  mm,	Y =   -70.461  mm,	Z =  -434.552  mm,
	W =     -.954 deg,	P =    22.924 deg,	R =      .993 deg
   GP2:
	UF : 1, UT : 1,
	J1=    45.000 deg,	J2=   180.000 deg
};
P[871]{
   GP1:
	UF : 1, UT : 1,		CONFIG : 'N U T, 0, 0, 0',
	X =  2191.595  mm,	Y =  -150.581  mm,	Z =  -435.156  mm,
	W =     -.956 deg,	P =    22.925 deg,	R =    22.595 deg
   GP2:
	UF : 1, UT : 1,
	J1=    45.000 deg,	J2=   180.000 deg
};
P[872]{
   GP1:
	UF : 1, UT : 1,		CONFIG : 'N U T, 0, 0, 0',
	X =  1531.039  mm,	Y =   -74.045  mm,	Z =   -60.070  mm,
	W =     1.185 deg,	P =   -23.204 deg,	R =    -8.287 deg
   GP2:
	UF : 1, UT : 1,
	J1=     0.000 deg,	J2=   180.000 deg
};
P[873]{
   GP1:
	UF : 1, UT : 1,		CONFIG : 'N U T, 0, 0, 0',
	X =  1531.995  mm,	Y =   -94.374  mm,	Z =   -60.791  mm,
	W =     1.176 deg,	P =   -23.207 deg,	R =    -8.281 deg
   GP2:
	UF : 1, UT : 1,
	J1=     0.000 deg,	J2=   180.000 deg
};
P[874]{
   GP1:
	UF : 1, UT : 1,		CONFIG : 'N U T, 0, 0, 0',
	X =  1532.795  mm,	Y =  -150.585  mm,	Z =   -61.433  mm,
	W =     1.185 deg,	P =   -23.200 deg,	R =    -8.290 deg
   GP2:
	UF : 1, UT : 1,
	J1=     0.000 deg,	J2=   180.000 deg
};
P[875]{
   GP1:
	UF : 1, UT : 1,		CONFIG : 'N U T, 0, 0, 0',
	X =  1532.399  mm,	Y =  -119.775  mm,	Z =   -61.224  mm,
	W =     1.182 deg,	P =   -23.203 deg,	R =    -8.289 deg
   GP2:
	UF : 1, UT : 1,
	J1=     0.000 deg,	J2=   180.000 deg
};
P[876]{
   GP1:
	UF : 1, UT : 1,		CONFIG : 'N U T, 0, 0, 0',
	X =  2377.991  mm,	Y =   -75.118  mm,	Z =   -21.967  mm,
	W =    40.518 deg,	P =    40.131 deg,	R =    23.486 deg
   GP2:
	UF : 1, UT : 1,
	J1=    80.000 deg,	J2=    90.000 deg
};
P[877]{
   GP1:
	UF : 1, UT : 1,		CONFIG : 'N U T, 0, 0, 0',
	X =  2373.865  mm,	Y =   -94.159  mm,	Z =   -21.772  mm,
	W =    40.517 deg,	P =    40.133 deg,	R =    54.911 deg
   GP2:
	UF : 1, UT : 1,
	J1=    80.000 deg,	J2=    90.000 deg
};
P[878]{
   GP1:
	UF : 1, UT : 1,		CONFIG : 'N U T, 0, 0, 0',
	X =  2374.227  mm,	Y =  -129.954  mm,	Z =   -20.479  mm,
	W =    40.518 deg,	P =    40.131 deg,	R =    54.925 deg
   GP2:
	UF : 1, UT : 1,
	J1=    80.000 deg,	J2=    90.000 deg
};
P[879]{
   GP1:
	UF : 1, UT : 1,		CONFIG : 'N U T, 0, 0, 0',
	X =  2375.496  mm,	Y =  -148.718  mm,	Z =   -20.852  mm,
	W =    39.922 deg,	P =    39.704 deg,	R =    81.922 deg
   GP2:
	UF : 1, UT : 1,
	J1=    80.000 deg,	J2=    90.000 deg
};
P[880]{
   GP1:
	UF : 1, UT : 1,		CONFIG : 'N U T, 0, 0, 0',
	X =  1673.244  mm,	Y =  -186.849  mm,	Z =   -12.723  mm,
	W =    38.562 deg,	P =    15.652 deg,	R =    22.711 deg
   GP2:
	UF : 1, UT : 1,
	J1=    90.000 deg,	J2=    90.000 deg
};
P[881]{
   GP1:
	UF : 1, UT : 1,		CONFIG : 'N U T, 0, 0, 0',
	X =  1704.281  mm,	Y =  -187.144  mm,	Z =   -10.891  mm,
	W =    38.570 deg,	P =    15.647 deg,	R =   -27.578 deg
   GP2:
	UF : 1, UT : 1,
	J1=    90.000 deg,	J2=    90.000 deg
};
P[882]{
   GP1:
	UF : 1, UT : 1,		CONFIG : 'N U T, 0, 0, 0',
	X =  1984.359  mm,	Y =  -186.916  mm,	Z =   -11.179  mm,
	W =    41.524 deg,	P =    13.967 deg,	R =   -26.862 deg
   GP2:
	UF : 1, UT : 1,
	J1=    90.000 deg,	J2=    90.000 deg
};
P[883]{
   GP1:
	UF : 1, UT : 1,		CONFIG : 'N U T, 0, 0, 0',
	X =  2000.913  mm,	Y =  -186.696  mm,	Z =   -10.347  mm,
	W =    38.528 deg,	P =    15.652 deg,	R =   -66.409 deg
   GP2:
	UF : 1, UT : 1,
	J1=    89.999 deg,	J2=    90.000 deg
};
P[884]{
   GP1:
	UF : 1, UT : 1,		CONFIG : 'N U T, 0, 0, 0',
	X =  2229.198  mm,	Y =    55.160  mm,	Z =     5.970  mm,
	W =    44.926 deg,	P =     3.034 deg,	R =    -3.042 deg
   GP2:
	UF : 1, UT : 1,
	J1=    90.000 deg,	J2=    90.000 deg
};
P[885]{
   GP1:
	UF : 1, UT : 1,		CONFIG : 'N U T, 0, 0, 0',
	X =  2267.476  mm,	Y =    55.786  mm,	Z =     6.601  mm,
	W =    44.923 deg,	P =     3.031 deg,	R =    -3.038 deg
   GP2:
	UF : 1, UT : 1,
	J1=    90.000 deg,	J2=    90.000 deg
};
P[886]{
   GP1:
	UF : 1, UT : 1,		CONFIG : 'N U T, 0, 0, 0',
	X =  2154.017  mm,	Y =    55.089  mm,	Z =    -2.879  mm,
	W =    44.921 deg,	P =     3.028 deg,	R =    -3.034 deg
   GP2:
	UF : 1, UT : 1,
	J1=    90.000 deg,	J2=    90.000 deg
};
P[887]{
   GP1:
	UF : 1, UT : 1,		CONFIG : 'N U T, 0, 0, 0',
	X =  2212.116  mm,	Y =    54.430  mm,	Z =    -1.611  mm,
	W =    44.924 deg,	P =     3.032 deg,	R =    -3.036 deg
   GP2:
	UF : 1, UT : 1,
	J1=    90.000 deg,	J2=    90.000 deg
};
P[888]{
   GP1:
	UF : 1, UT : 1,		CONFIG : 'N U T, 0, 0, 0',
	X =  2215.246  mm,	Y =    53.876  mm,	Z =     -.373  mm,
	W =    44.919 deg,	P =     3.026 deg,	R =   -14.186 deg
   GP2:
	UF : 1, UT : 1,
	J1=    90.000 deg,	J2=    90.000 deg
};
P[889]{
   GP1:
	UF : 1, UT : 1,		CONFIG : 'N U T, 0, 0, 0',
	X =  2118.129  mm,	Y =    53.365  mm,	Z =   -11.331  mm,
	W =    44.928 deg,	P =     3.034 deg,	R =     5.574 deg
   GP2:
	UF : 1, UT : 1,
	J1=    90.000 deg,	J2=    90.000 deg
};
P[890]{
   GP1:
	UF : 1, UT : 1,		CONFIG : 'N U T, 0, 0, 0',
	X =  2025.224  mm,	Y =    53.089  mm,	Z =   -11.323  mm,
	W =    44.928 deg,	P =     3.031 deg,	R =     5.581 deg
   GP2:
	UF : 1, UT : 1,
	J1=    90.000 deg,	J2=    90.000 deg
};
P[891]{
   GP1:
	UF : 1, UT : 1,		CONFIG : 'N U T, 0, 0, 0',
	X =  2012.630  mm,	Y =    53.107  mm,	Z =   -11.366  mm,
	W =    44.931 deg,	P =     3.043 deg,	R =    34.540 deg
   GP2:
	UF : 1, UT : 1,
	J1=    90.000 deg,	J2=    90.000 deg
};
P[892]{
   GP1:
	UF : 1, UT : 1,		CONFIG : 'N U T, 0, 0, 0',
	X =  1799.188  mm,	Y =    54.902  mm,	Z =    56.394  mm,
	W =    50.324 deg,	P =     2.539 deg,	R =    12.040 deg
   GP2:
	UF : 1, UT : 1,
	J1=    90.000 deg,	J2=    90.000 deg
};
P[893]{
   GP1:
	UF : 1, UT : 1,		CONFIG : 'N U T, 0, 0, 0',
	X =  1690.022  mm,	Y =    51.584  mm,	Z =    58.827  mm,
	W =    50.328 deg,	P =     2.543 deg,	R =    12.043 deg
   GP2:
	UF : 1, UT : 1,
	J1=    90.000 deg,	J2=    90.000 deg
};
P[894]{
   GP1:
	UF : 1, UT : 1,		CONFIG : 'N U T, 0, 0, 0',
	X =  1672.210  mm,	Y =    49.772  mm,	Z =    60.285  mm,
	W =    55.797 deg,	P =      .901 deg,	R =    26.090 deg
   GP2:
	UF : 1, UT : 1,
	J1=    90.000 deg,	J2=    90.000 deg
};
P[895]{
   GP1:
	UF : 1, UT : 1,		CONFIG : 'N U T, 0, 0, 0',
	X =  1820.347  mm,	Y =    53.166  mm,	Z =    58.863  mm,
	W =    52.751 deg,	P =    -4.416 deg,	R =     3.516 deg
   GP2:
	UF : 1, UT : 1,
	J1=    90.000 deg,	J2=    90.000 deg
};
P[896]{
   GP1:
	UF : 1, UT : 1,		CONFIG : 'N U T, 0, 0, 0',
	X =  1967.650  mm,	Y =    55.105  mm,	Z =    55.758  mm,
	W =    53.721 deg,	P =    -4.476 deg,	R =     3.442 deg
   GP2:
	UF : 1, UT : 1,
	J1=    90.000 deg,	J2=    90.000 deg
};
P[897]{
   GP1:
	UF : 1, UT : 1,		CONFIG : 'N U T, 0, 0, 0',
	X =  2000.056  mm,	Y =    51.972  mm,	Z =    58.502  mm,
	W =    52.868 deg,	P =   -12.268 deg,	R =   -23.051 deg
   GP2:
	UF : 1, UT : 1,
	J1=    90.000 deg,	J2=    90.000 deg
};
P[898]{
   GP1:
	UF : 1, UT : 1,		CONFIG : 'N U T, 0, 0, 0',
	X =  2229.180  mm,	Y =    66.099  mm,	Z =    -1.785  mm,
	W =   -44.609 deg,	P =    -6.680 deg,	R =    -6.730 deg
   GP2:
	UF : 1, UT : 1,
	J1=    90.000 deg,	J2=    90.000 deg
};
P[899]{
   GP1:
	UF : 1, UT : 1,		CONFIG : 'N U T, 0, 0, 0',
	X =  2266.839  mm,	Y =    67.302  mm,	Z =     -.064  mm,
	W =   -44.609 deg,	P =    -6.676 deg,	R =    -6.726 deg
   GP2:
	UF : 1, UT : 1,
	J1=    90.000 deg,	J2=    90.000 deg
};
P[900]{
   GP1:
	UF : 1, UT : 1,		CONFIG : 'N U T, 0, 0, 0',
	X =  2139.677  mm,	Y =    66.559  mm,	Z =    -8.353  mm,
	W =   -44.605 deg,	P =    -6.678 deg,	R =    -6.724 deg
   GP2:
	UF : 1, UT : 1,
	J1=    90.000 deg,	J2=    90.000 deg
};
P[901]{
   GP1:
	UF : 1, UT : 1,		CONFIG : 'N U T, 0, 0, 0',
	X =  2207.201  mm,	Y =    67.923  mm,	Z =    -7.410  mm,
	W =   -44.606 deg,	P =    -6.676 deg,	R =    -6.723 deg
   GP2:
	UF : 1, UT : 1,
	J1=    90.000 deg,	J2=    90.000 deg
};
P[902]{
   GP1:
	UF : 1, UT : 1,		CONFIG : 'N U T, 0, 0, 0',
	X =  2213.314  mm,	Y =    66.559  mm,	Z =    -7.780  mm,
	W =   -44.607 deg,	P =    -6.680 deg,	R =     6.845 deg
   GP2:
	UF : 1, UT : 1,
	J1=    90.000 deg,	J2=    90.000 deg
};
P[903]{
   GP1:
	UF : 1, UT : 1,		CONFIG : 'N U T, 0, 0, 0',
	X =  1993.335  mm,	Y =    66.632  mm,	Z =   -18.063  mm,
	W =   -44.598 deg,	P =    -6.687 deg,	R =    -3.028 deg
   GP2:
	UF : 1, UT : 1,
	J1=    90.000 deg,	J2=    90.000 deg
};
P[904]{
   GP1:
	UF : 1, UT : 1,		CONFIG : 'N U T, 0, 0, 0',
	X =  2106.177  mm,	Y =    68.196  mm,	Z =   -16.279  mm,
	W =   -44.610 deg,	P =    -6.676 deg,	R =    -3.020 deg
   GP2:
	UF : 1, UT : 1,
	J1=    90.000 deg,	J2=    90.000 deg
};
P[905]{
   GP1:
	UF : 1, UT : 1,		CONFIG : 'N U T, 0, 0, 0',
	X =  2115.669  mm,	Y =    68.079  mm,	Z =   -12.688  mm,
	W =   -42.116 deg,	P =   -17.568 deg,	R =    21.832 deg
   GP2:
	UF : 1, UT : 1,
	J1=    90.000 deg,	J2=    90.000 deg
};
P[906]{
   GP1:
	UF : 1, UT : 1,		CONFIG : 'N U T, 0, 0, 0',
	X =  2008.751  mm,	Y =   102.079  mm,	Z =   -12.082  mm,
	W =   -45.253 deg,	P =    -8.453 deg,	R =  -108.141 deg
   GP2:
	UF : 1, UT : 1,
	J1=    90.000 deg,	J2=   100.000 deg
};
P[907]{
   GP1:
	UF : 1, UT : 1,		CONFIG : 'N U T, 0, 0, 0',
	X =  2009.223  mm,	Y =  -122.001  mm,	Z =   -48.481  mm,
	W =   -45.248 deg,	P =    -8.452 deg,	R =   -86.326 deg
   GP2:
	UF : 1, UT : 1,
	J1=    90.000 deg,	J2=   100.000 deg
};
P[908]{
   GP1:
	UF : 1, UT : 1,		CONFIG : 'N U T, 0, 0, 0',
	X =  2756.457  mm,	Y =   175.047  mm,	Z =   183.225  mm,
	W =     2.780 deg,	P =    -7.669 deg,	R =   -18.458 deg
   GP2:
	UF : 1, UT : 1,
	J1=    90.000 deg,	J2=   135.000 deg
};
P[909]{
   GP1:
	UF : 1, UT : 1,		CONFIG : 'N U T, 0, 0, 0',
	X =  2866.579  mm,	Y =   178.189  mm,	Z =   188.861  mm,
	W =     9.502 deg,	P =   -26.582 deg,	R =   -20.495 deg
   GP2:
	UF : 1, UT : 1,
	J1=    89.999 deg,	J2=   135.000 deg
};
P[910]{
   GP1:
	UF : 1, UT : 1,		CONFIG : 'N U T, 0, 0, 0',
	X =  2382.254  mm,	Y =   277.346  mm,	Z =    92.106  mm,
	W =     1.846 deg,	P =     -.179 deg,	R =      .947 deg
   GP2:
	UF : 1, UT : 1,
	J1=    90.000 deg,	J2=   135.000 deg
};
P[911]{
   GP1:
	UF : 1, UT : 1,		CONFIG : 'N U T, 0, 0, 0',
	X =  2756.953  mm,	Y =   278.563  mm,	Z =    92.649  mm,
	W =     1.723 deg,	P =    -7.244 deg,	R =      .958 deg
   GP2:
	UF : 1, UT : 1,
	J1=    90.000 deg,	J2=   135.000 deg
};
P[912]{
   GP1:
	UF : 1, UT : 1,		CONFIG : 'N U T, 0, 0, 0',
	X =  2079.674  mm,	Y =   119.684  mm,	Z =   -13.503  mm,
	W =    37.938 deg,	P =    17.393 deg,	R =   -97.677 deg
   GP2:
	UF : 1, UT : 1,
	J1=    90.000 deg,	J2=    90.000 deg
};
P[913]{
   GP1:
	UF : 1, UT : 1,		CONFIG : 'N U T, 0, 0, 0',
	X =  2107.541  mm,	Y =    91.774  mm,	Z =   -12.232  mm,
	W =    37.933 deg,	P =    17.391 deg,	R =  -104.290 deg
   GP2:
	UF : 1, UT : 1,
	J1=    90.000 deg,	J2=    90.000 deg
};
P[914]{
   GP1:
	UF : 1, UT : 1,		CONFIG : 'N U T, 0, 0, -1',
	X =  2123.963  mm,	Y =    74.328  mm,	Z =    -9.686  mm,
	W =    40.829 deg,	P =    19.041 deg,	R =  -124.269 deg
   GP2:
	UF : 1, UT : 1,
	J1=    90.000 deg,	J2=    90.000 deg
};
P[915]{
   GP1:
	UF : 1, UT : 1,		CONFIG : 'N U T, 0, 0, 0',
	X =  1688.578  mm,	Y =    68.430  mm,	Z =   -18.303  mm,
	W =   -42.811 deg,	P =    15.445 deg,	R =    16.037 deg
   GP2:
	UF : 1, UT : 1,
	J1=    90.000 deg,	J2=    90.000 deg
};
P[916]{
   GP1:
	UF : 1, UT : 1,		CONFIG : 'N U T, 0, 0, 0',
	X =  1651.189  mm,	Y =    68.384  mm,	Z =   -18.170  mm,
	W =   -42.811 deg,	P =    15.445 deg,	R =    16.039 deg
   GP2:
	UF : 1, UT : 1,
	J1=    90.000 deg,	J2=    90.000 deg
};
P[917]{
   GP1:
	UF : 1, UT : 1,		CONFIG : 'N U T, 0, 0, 0',
	X =  1641.486  mm,	Y =    69.984  mm,	Z =   -18.017  mm,
	W =   -42.802 deg,	P =    15.441 deg,	R =    -7.970 deg
   GP2:
	UF : 1, UT : 1,
	J1=    90.000 deg,	J2=    90.000 deg
};
P[918]{
   GP1:
	UF : 1, UT : 1,		CONFIG : 'N U T, 0, 0, 0',
	X =  1635.303  mm,	Y =    72.574  mm,	Z =   -19.890  mm,
	W =   -38.580 deg,	P =    25.212 deg,	R =   -16.906 deg
   GP2:
	UF : 1, UT : 1,
	J1=    90.000 deg,	J2=    90.000 deg
};
P[919]{
   GP1:
	UF : 1, UT : 1,		CONFIG : 'N U T, 0, 0, 0',
	X =  1607.511  mm,	Y =   100.945  mm,	Z =   -20.220  mm,
	W =   -38.581 deg,	P =    25.213 deg,	R =   -16.910 deg
   GP2:
	UF : 1, UT : 1,
	J1=    90.000 deg,	J2=    90.000 deg
};
P[920]{
   GP1:
	UF : 1, UT : 1,		CONFIG : 'N U T, 0, 0, 0',
	X =  1584.434  mm,	Y =   111.509  mm,	Z =   -19.223  mm,
	W =   -44.998 deg,	P =    -3.171 deg,	R =      .428 deg
   GP2:
	UF : 1, UT : 1,
	J1=    90.000 deg,	J2=    90.000 deg
};
P[921]{
   GP1:
	UF : 1, UT : 1,		CONFIG : 'N U T, 0, 0, 0',
	X =  1565.857  mm,	Y =    86.604  mm,	Z =   -16.661  mm,
	W =   -45.448 deg,	P =    19.946 deg,	R =    98.978 deg
   GP2:
	UF : 1, UT : 1,
	J1=    90.000 deg,	J2=    90.000 deg
};
P[922]{
   GP1:
	UF : 1, UT : 1,		CONFIG : 'N U T, 0, 0, 0',
	X =  1561.980  mm,	Y =    43.412  mm,	Z =   -17.393  mm,
	W =   -45.341 deg,	P =    20.071 deg,	R =    97.877 deg
   GP2:
	UF : 1, UT : 1,
	J1=    90.000 deg,	J2=    90.000 deg
};
P[923]{
   GP1:
	UF : 1, UT : 1,		CONFIG : 'N U T, 0, 0, 0',
	X =  1557.455  mm,	Y =    34.734  mm,	Z =   -14.659  mm,
	W =   -41.212 deg,	P =    19.951 deg,	R =    68.903 deg
   GP2:
	UF : 1, UT : 1,
	J1=    90.000 deg,	J2=    90.000 deg
};
P[924]{
   GP1:
	UF : 1, UT : 1,		CONFIG : 'N U T, 0, 0, 0',
	X =  1551.432  mm,	Y =    29.710  mm,	Z =   -18.261  mm,
	W =   -41.212 deg,	P =    19.944 deg,	R =    34.864 deg
   GP2:
	UF : 1, UT : 1,
	J1=    90.000 deg,	J2=    90.000 deg
};
P[925]{
   GP1:
	UF : 1, UT : 1,		CONFIG : 'N U T, 0, 0, 0',
	X =  1545.443  mm,	Y =    27.978  mm,	Z =   -18.518  mm,
	W =   -41.206 deg,	P =    19.937 deg,	R =    34.859 deg
   GP2:
	UF : 1, UT : 1,
	J1=    90.000 deg,	J2=    90.000 deg
};
P[926]{
   GP1:
	UF : 1, UT : 1,		CONFIG : 'N U T, 0, 0, 0',
	X =  2865.227  mm,	Y =  1437.901  mm,	Z =    -5.229  mm,
	W =     -.178 deg,	P =    -1.186 deg,	R =    26.508 deg
   GP2:
	UF : 1, UT : 1,
	J1=    90.000 deg,	J2=    90.000 deg
};
P[927]{
   GP1:
	UF : 1, UT : 1,		CONFIG : 'N U T, 0, 0, 0',
	X =  2865.228  mm,	Y =  1421.330  mm,	Z =    -5.229  mm,
	W =     -.178 deg,	P =    -1.186 deg,	R =    26.508 deg
   GP2:
	UF : 1, UT : 1,
	J1=    90.000 deg,	J2=    90.000 deg
};
P[928]{
   GP1:
	UF : 1, UT : 1,		CONFIG : 'N U T, 0, 0, 0',
	X =  2850.371  mm,	Y =  1421.330  mm,	Z =    -5.228  mm,
	W =     -.178 deg,	P =    -1.186 deg,	R =    26.508 deg
   GP2:
	UF : 1, UT : 1,
	J1=    90.000 deg,	J2=    90.000 deg
};
P[929]{
   GP1:
	UF : 1, UT : 1,		CONFIG : 'N U T, 0, 0, 0',
	X =  2850.370  mm,	Y =  1421.329  mm,	Z =     -.942  mm,
	W =     -.178 deg,	P =    -1.186 deg,	R =    26.508 deg
   GP2:
	UF : 1, UT : 1,
	J1=    90.000 deg,	J2=    90.000 deg
};
P[930]{
   GP1:
	UF : 1, UT : 1,		CONFIG : 'N U T, 0, 0, 0',
	X =  2850.129  mm,	Y =  1437.623  mm,	Z =    -5.153  mm,
	W =     -.178 deg,	P =    -1.186 deg,	R =    26.509 deg
   GP2:
	UF : 1, UT : 1,
	J1=    90.000 deg,	J2=    90.000 deg
};
P[931]{
   GP1:
	UF : 1, UT : 1,		CONFIG : 'N U T, 0, 0, 0',
	X =  2850.129  mm,	Y =  1437.623  mm,	Z =     -.867  mm,
	W =     -.178 deg,	P =    -1.186 deg,	R =    26.509 deg
   GP2:
	UF : 1, UT : 1,
	J1=    90.000 deg,	J2=    90.000 deg
};
P[932]{
   GP1:
	UF : 1, UT : 1,		CONFIG : 'N U T, 0, 0, 1',
	X =  1661.474  mm,	Y =  -211.430  mm,	Z =   -14.467  mm,
	W =   -32.923 deg,	P =    29.352 deg,	R =   129.298 deg
   GP2:
	UF : 1, UT : 1,
	J1=    90.000 deg,	J2=    90.000 deg
};
P[933]{
   GP1:
	UF : 1, UT : 1,		CONFIG : 'N U T, 0, 0, 1',
	X =  1661.456  mm,	Y =    27.029  mm,	Z =   -15.234  mm,
	W =   -34.235 deg,	P =    30.074 deg,	R =   141.357 deg
   GP2:
	UF : 1, UT : 1,
	J1=    90.000 deg,	J2=    90.000 deg
};
P[934]{
   GP1:
	UF : 1, UT : 1,		CONFIG : 'N U T, 0, 0, 0',
	X =  2356.583  mm,	Y =  -166.791  mm,	Z =    -1.143  mm,
	W =    44.579 deg,	P =     6.896 deg,	R =    -6.948 deg
   GP2:
	UF : 1, UT : 1,
	J1=    90.000 deg,	J2=    90.000 deg
};
P[935]{
   GP1:
	UF : 1, UT : 1,		CONFIG : 'N U T, 0, 0, 0',
	X =  2528.956  mm,	Y =  -162.655  mm,	Z =     -.745  mm,
	W =    44.582 deg,	P =     6.894 deg,	R =    -6.935 deg
   GP2:
	UF : 1, UT : 1,
	J1=    90.000 deg,	J2=    90.000 deg
};
P[936]{
   GP1:
	UF : 1, UT : 1,		CONFIG : 'N U T, 0, 0, 0',
	X =  2357.492  mm,	Y =   -79.748  mm,	Z =     -.449  mm,
	W =    43.253 deg,	P =    13.899 deg,	R =   -18.619 deg
   GP2:
	UF : 1, UT : 1,
	J1=    90.000 deg,	J2=    90.000 deg
};
P[937]{
   GP1:
	UF : 1, UT : 1,		CONFIG : 'N U T, 0, 0, 0',
	X =  2403.170  mm,	Y =   -77.561  mm,	Z =     -.153  mm,
	W =    43.247 deg,	P =    13.894 deg,	R =   -18.614 deg
   GP2:
	UF : 1, UT : 1,
	J1=    90.000 deg,	J2=    90.000 deg
};
P[938]{
   GP1:
	UF : 1, UT : 1,		CONFIG : 'N U T, 0, 0, 0',
	X =  2425.265  mm,	Y =   -75.847  mm,	Z =     -.682  mm,
	W =    42.932 deg,	P =    13.800 deg,	R =   -51.812 deg
   GP2:
	UF : 1, UT : 1,
	J1=    89.994 deg,	J2=    90.001 deg
};
P[939]{
   GP1:
	UF : 1, UT : 1,		CONFIG : 'N U T, 0, 0, 0',
	X =  1683.325  mm,	Y =   473.158  mm,	Z =   835.968  mm,
	W =    39.872 deg,	P =   -22.882 deg,	R =   -65.015 deg
   GP2:
	UF : 1, UT : 1,
	J1=   -90.000 deg,	J2=   -90.000 deg
};
P[940]{
   GP1:
	UF : 1, UT : 1,		CONFIG : 'N U T, 0, 0, 0',
	X =  1684.315  mm,	Y =   491.221  mm,	Z =   835.551  mm,
	W =    39.874 deg,	P =   -22.882 deg,	R =   -65.014 deg
   GP2:
	UF : 1, UT : 1,
	J1=   -90.000 deg,	J2=   -90.000 deg
};
P[941]{
   GP1:
	UF : 1, UT : 1,		CONFIG : 'N U T, 0, 0, 0',
	X =  1684.342  mm,	Y =   498.399  mm,	Z =   835.965  mm,
	W =    39.869 deg,	P =   -22.881 deg,	R =   -69.837 deg
   GP2:
	UF : 1, UT : 1,
	J1=   -90.000 deg,	J2=   -90.000 deg
};
P[942]{
   GP1:
	UF : 1, UT : 1,		CONFIG : 'N U T, 0, 0, 0',
	X =  1686.294  mm,	Y =   502.192  mm,	Z =   835.782  mm,
	W =    39.867 deg,	P =   -22.881 deg,	R =   -70.971 deg
   GP2:
	UF : 1, UT : 1,
	J1=   -90.000 deg,	J2=   -90.000 deg
};
P[943]{
   GP1:
	UF : 1, UT : 1,		CONFIG : 'N U T, 0, 0, 0',
	X =  1709.542  mm,	Y =   572.021  mm,	Z =   833.650  mm,
	W =    39.889 deg,	P =   -22.872 deg,	R =   -70.981 deg
   GP2:
	UF : 1, UT : 1,
	J1=   -90.000 deg,	J2=   -90.000 deg
};
P[944]{
   GP1:
	UF : 1, UT : 1,		CONFIG : 'N U T, 0, 0, 0',
	X =  1709.635  mm,	Y =   574.784  mm,	Z =   834.621  mm,
	W =    39.875 deg,	P =   -22.876 deg,	R =   -74.849 deg
   GP2:
	UF : 1, UT : 1,
	J1=   -90.000 deg,	J2=   -90.000 deg
};
P[945]{
   GP1:
	UF : 1, UT : 1,		CONFIG : 'N U T, 0, 0, 0',
	X =  1712.926  mm,	Y =   578.115  mm,	Z =   833.070  mm,
	W =    39.876 deg,	P =   -22.873 deg,	R =   -82.539 deg
   GP2:
	UF : 1, UT : 1,
	J1=   -90.000 deg,	J2=   -90.000 deg
};
P[946]{
   GP1:
	UF : 1, UT : 1,		CONFIG : 'N U T, 0, 0, 0',
	X =  1847.977  mm,	Y =   837.117  mm,	Z =   835.341  mm,
	W =    14.308 deg,	P =   -43.040 deg,	R =   -40.623 deg
   GP2:
	UF : 1, UT : 1,
	J1=   -89.991 deg,	J2=   -89.999 deg
};
P[947]{
   GP1:
	UF : 1, UT : 1,		CONFIG : 'N U T, 0, 0, 0',
	X =  1705.072  mm,	Y =   434.306  mm,	Z =   834.623  mm,
	W =    43.039 deg,	P =   -14.376 deg,	R =   -45.080 deg
   GP2:
	UF : 1, UT : 1,
	J1=   -90.000 deg,	J2=   -90.000 deg
};
P[948]{
   GP1:
	UF : 1, UT : 1,		CONFIG : 'N U T, 0, 0, 0',
	X =  1837.222  mm,	Y =   282.936  mm,	Z =   837.197  mm,
	W =    43.048 deg,	P =   -14.367 deg,	R =   -45.080 deg
   GP2:
	UF : 1, UT : 1,
	J1=   -90.000 deg,	J2=   -90.000 deg
};
P[949]{
   GP1:
	UF : 1, UT : 1,		CONFIG : 'N U T, 0, 0, 0',
	X =  1846.282  mm,	Y =   274.844  mm,	Z =   836.456  mm,
	W =    43.043 deg,	P =   -14.373 deg,	R =   -42.869 deg
   GP2:
	UF : 1, UT : 1,
	J1=   -90.000 deg,	J2=   -90.000 deg
};
P[950]{
   GP1:
	UF : 1, UT : 1,		CONFIG : 'N U T, 0, 0, 0',
	X =  1858.284  mm,	Y =   264.264  mm,	Z =   837.590  mm,
	W =    43.040 deg,	P =   -14.375 deg,	R =   -40.827 deg
   GP2:
	UF : 1, UT : 1,
	J1=   -90.000 deg,	J2=   -90.000 deg
};
P[951]{
   GP1:
	UF : 1, UT : 1,		CONFIG : 'N U T, 0, 0, 0',
	X =  1921.924  mm,	Y =   216.710  mm,	Z =   837.742  mm,
	W =    43.043 deg,	P =   -14.374 deg,	R =   -40.827 deg
   GP2:
	UF : 1, UT : 1,
	J1=   -90.000 deg,	J2=   -90.000 deg
};
P[952]{
   GP1:
	UF : 1, UT : 1,		CONFIG : 'N U T, 0, 0, 0',
	X =  1682.193  mm,	Y =  -453.390  mm,	Z =   837.036  mm,
	W =   -28.324 deg,	P =   -37.469 deg,	R =    36.656 deg
   GP2:
	UF : 1, UT : 1,
	J1=   -90.000 deg,	J2=    90.000 deg
};
P[953]{
   GP1:
	UF : 1, UT : 1,		CONFIG : 'N U T, 0, 0, 0',
	X =  1681.929  mm,	Y =  -469.569  mm,	Z =   837.938  mm,
	W =   -28.311 deg,	P =   -37.472 deg,	R =    36.643 deg
   GP2:
	UF : 1, UT : 1,
	J1=   -90.000 deg,	J2=    90.000 deg
};
P[954]{
   GP1:
	UF : 1, UT : 1,		CONFIG : 'N U T, 0, 0, 0',
	X =  1682.868  mm,	Y =  -474.172  mm,	Z =   837.920  mm,
	W =   -28.319 deg,	P =   -37.466 deg,	R =    39.717 deg
   GP2:
	UF : 1, UT : 1,
	J1=   -90.000 deg,	J2=    90.000 deg
};
P[955]{
   GP1:
	UF : 1, UT : 1,		CONFIG : 'N U T, 0, 0, 0',
	X =  1683.234  mm,	Y =  -476.970  mm,	Z =   837.454  mm,
	W =   -28.320 deg,	P =   -37.464 deg,	R =    41.169 deg
   GP2:
	UF : 1, UT : 1,
	J1=   -90.000 deg,	J2=    90.000 deg
};
P[956]{
   GP1:
	UF : 1, UT : 1,		CONFIG : 'N U T, 0, 0, 0',
	X =  1705.800  mm,	Y =  -547.787  mm,	Z =   836.670  mm,
	W =   -28.304 deg,	P =   -37.472 deg,	R =    41.151 deg
   GP2:
	UF : 1, UT : 1,
	J1=   -90.000 deg,	J2=    90.000 deg
};
P[957]{
   GP1:
	UF : 1, UT : 1,		CONFIG : 'N U T, 0, 0, 0',
	X =  1708.265  mm,	Y =  -551.949  mm,	Z =   836.333  mm,
	W =   -28.320 deg,	P =   -37.465 deg,	R =    48.503 deg
   GP2:
	UF : 1, UT : 1,
	J1=   -90.000 deg,	J2=    90.000 deg
};
P[958]{
   GP1:
	UF : 1, UT : 1,		CONFIG : 'N U T, 0, 0, 0',
	X =  1711.157  mm,	Y =  -557.289  mm,	Z =   835.170  mm,
	W =   -28.318 deg,	P =   -37.465 deg,	R =    55.395 deg
   GP2:
	UF : 1, UT : 1,
	J1=   -90.000 deg,	J2=    90.000 deg
};
P[959]{
   GP1:
	UF : 1, UT : 1,		CONFIG : 'N U T, 0, 0, 0',
	X =  1849.295  mm,	Y =  -818.144  mm,	Z =   836.002  mm,
	W =   -28.326 deg,	P =   -37.469 deg,	R =    50.637 deg
   GP2:
	UF : 1, UT : 1,
	J1=   -90.000 deg,	J2=    90.000 deg
};
P[960]{
   GP1:
	UF : 1, UT : 1,		CONFIG : 'N U T, 0, 0, 0',
	X =  1704.432  mm,	Y =  -414.901  mm,	Z =   836.550  mm,
	W =   -39.458 deg,	P =    -8.332 deg,	R =    42.662 deg
   GP2:
	UF : 1, UT : 1,
	J1=   -90.000 deg,	J2=    90.000 deg
};
P[961]{
   GP1:
	UF : 1, UT : 1,		CONFIG : 'N U T, 0, 0, 0',
	X =  1836.725  mm,	Y =  -261.130  mm,	Z =   837.566  mm,
	W =   -39.460 deg,	P =    -8.334 deg,	R =    42.657 deg
   GP2:
	UF : 1, UT : 1,
	J1=   -90.000 deg,	J2=    90.000 deg
};
P[962]{
   GP1:
	UF : 1, UT : 1,		CONFIG : 'N U T, 0, 0, 0',
	X =  1847.154  mm,	Y =  -250.558  mm,	Z =   837.780  mm,
	W =   -39.460 deg,	P =    -8.334 deg,	R =    38.620 deg
   GP2:
	UF : 1, UT : 1,
	J1=   -90.000 deg,	J2=    90.000 deg
};
P[963]{
   GP1:
	UF : 1, UT : 1,		CONFIG : 'N U T, 0, 0, 0',
	X =  1865.972  mm,	Y =  -238.338  mm,	Z =   836.303  mm,
	W =   -39.464 deg,	P =    -8.329 deg,	R =    41.376 deg
   GP2:
	UF : 1, UT : 1,
	J1=   -90.000 deg,	J2=    90.000 deg
};
P[964]{
   GP1:
	UF : 1, UT : 1,		CONFIG : 'N U T, 0, 0, 0',
	X =  1936.009  mm,	Y =  -184.129  mm,	Z =   835.922  mm,
	W =   -39.460 deg,	P =    -8.334 deg,	R =    45.243 deg
   GP2:
	UF : 1, UT : 1,
	J1=   -90.000 deg,	J2=    90.000 deg
};
P[965]{
   GP1:
	UF : 1, UT : 1,		CONFIG : 'N U T, 0, 0, 0',
	X =  2332.738  mm,	Y =   -47.271  mm,	Z =   843.561  mm,
	W =     4.734 deg,	P =    44.798 deg,	R =    66.699 deg
   GP2:
	UF : 1, UT : 1,
	J1=    90.000 deg,	J2=    90.000 deg
};
P[966]{
   GP1:
	UF : 1, UT : 1,		CONFIG : 'N U T, 0, 0, 0',
	X =  2397.915  mm,	Y =   -81.738  mm,	Z =   843.540  mm,
	W =     4.740 deg,	P =    44.803 deg,	R =    66.701 deg
   GP2:
	UF : 1, UT : 1,
	J1=    90.000 deg,	J2=    90.000 deg
};
P[967]{
   GP1:
	UF : 1, UT : 1,		CONFIG : 'N U T, 0, 0, 0',
	X =  2392.544  mm,	Y =  -101.513  mm,	Z =   844.600  mm,
	W =   -19.423 deg,	P =    41.434 deg,	R =   -56.042 deg
   GP2:
	UF : 1, UT : 1,
	J1=    90.000 deg,	J2=    90.000 deg
};
P[968]{
   GP1:
	UF : 1, UT : 1,		CONFIG : 'N U T, 0, 0, 0',
	X =  2404.369  mm,	Y =   -81.730  mm,	Z =   844.555  mm,
	W =   -19.420 deg,	P =    41.429 deg,	R =   -56.056 deg
   GP2:
	UF : 1, UT : 1,
	J1=    90.000 deg,	J2=    90.000 deg
};
P[969]{
   GP1:
	UF : 1, UT : 1,		CONFIG : 'N U T, 0, 0, 0',
	X =  2328.544  mm,	Y =   -68.370  mm,	Z =   846.428  mm,
	W =    34.013 deg,	P =    31.443 deg,	R =   -66.602 deg
   GP2:
	UF : 1, UT : 1,
	J1=    90.000 deg,	J2=    90.000 deg
};
P[970]{
   GP1:
	UF : 1, UT : 1,		CONFIG : 'N U T, 0, 0, 0',
	X =  2393.286  mm,	Y =  -101.982  mm,	Z =   846.571  mm,
	W =    34.017 deg,	P =    31.444 deg,	R =   -66.601 deg
   GP2:
	UF : 1, UT : 1,
	J1=    90.000 deg,	J2=    90.000 deg
};
P[971]{
   GP1:
	UF : 1, UT : 1,		CONFIG : 'N U T, 0, 0, 0',
	X =  2528.546  mm,	Y =   -75.301  mm,	Z =   -25.347  mm,
	W =   -31.378 deg,	P =   -16.422 deg,	R =   -28.757 deg
   GP2:
	UF : 1, UT : 1,
	J1=    90.000 deg,	J2=   100.000 deg
};
P[972]{
   GP1:
	UF : 1, UT : 1,		CONFIG : 'N U T, 0, 0, 0',
	X =  2478.819  mm,	Y =   -77.760  mm,	Z =   -27.432  mm,
	W =   -25.030 deg,	P =   -25.322 deg,	R =   -46.368 deg
   GP2:
	UF : 1, UT : 1,
	J1=    90.000 deg,	J2=   100.000 deg
};
P[973]{
   GP1:
	UF : 1, UT : 1,		CONFIG : 'N U T, 0, 0, 0',
	X =  2453.018  mm,	Y =   -75.007  mm,	Z =   -22.167  mm,
	W =   -25.030 deg,	P =   -25.320 deg,	R =   -79.891 deg
   GP2:
	UF : 1, UT : 1,
	J1=    90.000 deg,	J2=   100.000 deg
};
P[974]{
   GP1:
	UF : 1, UT : 1,		CONFIG : 'N U T, 0, 0, 0',
	X =  2355.417  mm,	Y =   -77.872  mm,	Z =   -26.021  mm,
	W =   -31.933 deg,	P =   -15.149 deg,	R =   -17.048 deg
   GP2:
	UF : 1, UT : 1,
	J1=    90.000 deg,	J2=   100.000 deg
};
P[975]{
   GP1:
	UF : 1, UT : 1,		CONFIG : 'N U T, 0, 0, 0',
	X =  2405.871  mm,	Y =   -77.687  mm,	Z =   -25.824  mm,
	W =   -31.936 deg,	P =   -15.140 deg,	R =   -17.039 deg
   GP2:
	UF : 1, UT : 1,
	J1=    90.000 deg,	J2=   100.000 deg
};
P[976]{
   GP1:
	UF : 1, UT : 1,		CONFIG : 'N U T, 0, 0, 0',
	X =  2425.431  mm,	Y =   -74.422  mm,	Z =   -19.845  mm,
	W =   -21.656 deg,	P =   -28.186 deg,	R =   -20.809 deg
   GP2:
	UF : 1, UT : 1,
	J1=    90.000 deg,	J2=   100.000 deg
};
P[977]{
   GP1:
	UF : 1, UT : 1,		CONFIG : 'N U T, 0, 0, -1',
	X =  2131.448  mm,	Y =   167.383  mm,	Z =   837.718  mm,
	W =     2.978 deg,	P =    35.508 deg,	R =   160.120 deg
   GP2:
	UF : 1, UT : 1,
	J1=    90.000 deg,	J2=    90.000 deg
};
P[978]{
   GP1:
	UF : 1, UT : 1,		CONFIG : 'N U T, 0, 0, -1',
	X =  2138.426  mm,	Y =   185.708  mm,	Z =   836.262  mm,
	W =     2.984 deg,	P =    35.512 deg,	R =   160.108 deg
   GP2:
	UF : 1, UT : 1,
	J1=    90.000 deg,	J2=    90.000 deg
};
P[979]{
   GP1:
	UF : 1, UT : 1,		CONFIG : 'N U T, 0, 0, 0',
	X =  2123.406  mm,	Y =   217.744  mm,	Z =   837.111  mm,
	W =     2.989 deg,	P =    35.514 deg,	R =  -100.158 deg
   GP2:
	UF : 1, UT : 1,
	J1=    90.000 deg,	J2=    90.000 deg
};
P[980]{
   GP1:
	UF : 1, UT : 1,		CONFIG : 'N U T, 0, 0, 0',
	X =  2092.958  mm,	Y =   207.232  mm,	Z =   834.589  mm,
	W =     2.994 deg,	P =    35.514 deg,	R =   -13.063 deg
   GP2:
	UF : 1, UT : 1,
	J1=    90.000 deg,	J2=    90.000 deg
};
P[981]{
   GP1:
	UF : 1, UT : 1,		CONFIG : 'N U T, 0, 0, 0',
	X =  2078.138  mm,	Y =   163.139  mm,	Z =   834.542  mm,
	W =     2.985 deg,	P =    35.519 deg,	R =   -13.063 deg
   GP2:
	UF : 1, UT : 1,
	J1=    90.000 deg,	J2=    90.000 deg
};
P[982]{
   GP1:
	UF : 1, UT : 1,		CONFIG : 'N U T, 0, 0, 0',
	X =  2096.759  mm,	Y =   132.279  mm,	Z =   836.139  mm,
	W =     2.980 deg,	P =    35.506 deg,	R =    77.138 deg
   GP2:
	UF : 1, UT : 1,
	J1=    90.000 deg,	J2=    90.000 deg
};
P[983]{
   GP1:
	UF : 1, UT : 1,		CONFIG : 'N U T, 0, 0, 0',
	X =  2125.080  mm,	Y =   144.467  mm,	Z =   837.660  mm,
	W =     2.985 deg,	P =    35.516 deg,	R =   159.524 deg
   GP2:
	UF : 1, UT : 1,
	J1=    90.000 deg,	J2=    90.000 deg
};
P[984]{
   GP1:
	UF : 1, UT : 1,		CONFIG : 'N U T, 0, 0, 0',
	X =  2131.538  mm,	Y =   166.438  mm,	Z =   838.726  mm,
	W =     2.983 deg,	P =    35.509 deg,	R =   159.515 deg
   GP2:
	UF : 1, UT : 1,
	J1=    90.000 deg,	J2=    90.000 deg
};
P[985]{
   GP1:
	UF : 1, UT : 1,		CONFIG : 'N U T, 0, 0, 0',
	X =  2111.672  mm,	Y =   237.739  mm,	Z =   836.183  mm,
	W =    -2.356 deg,	P =    42.845 deg,	R =    86.535 deg
   GP2:
	UF : 1, UT : 1,
	J1=    90.000 deg,	J2=    90.000 deg
};
P[986]{
   GP1:
	UF : 1, UT : 1,		CONFIG : 'N U T, 0, 0, 0',
	X =  2190.874  mm,	Y =   237.707  mm,	Z =   836.167  mm,
	W =    -2.351 deg,	P =    42.846 deg,	R =    86.540 deg
   GP2:
	UF : 1, UT : 1,
	J1=    90.000 deg,	J2=    90.000 deg
};
P[987]{
   GP1:
	UF : 1, UT : 1,		CONFIG : 'N U T, 0, 0, 0',
	X =  2202.749  mm,	Y =   236.200  mm,	Z =   835.913  mm,
	W =    -2.491 deg,	P =    44.296 deg,	R =    56.657 deg
   GP2:
	UF : 1, UT : 1,
	J1=    90.000 deg,	J2=    90.000 deg
};
P[988]{
   GP1:
	UF : 1, UT : 1,		CONFIG : 'N U T, 0, 0, 0',
	X =  2210.456  mm,	Y =   232.643  mm,	Z =   837.248  mm,
	W =      .034 deg,	P =    44.146 deg,	R =    40.391 deg
   GP2:
	UF : 1, UT : 1,
	J1=    90.000 deg,	J2=    90.000 deg
};
P[989]{
   GP1:
	UF : 1, UT : 1,		CONFIG : 'N U T, 0, 0, 0',
	X =  2435.847  mm,	Y =   -25.240  mm,	Z =   836.935  mm,
	W =     -.127 deg,	P =    43.812 deg,	R =    45.343 deg
   GP2:
	UF : 1, UT : 1,
	J1=    90.000 deg,	J2=    90.000 deg
};
P[990]{
   GP1:
	UF : 1, UT : 1,		CONFIG : 'N U T, 0, 0, 0',
	X =  2452.948  mm,	Y =   -41.289  mm,	Z =   836.917  mm,
	W =      .173 deg,	P =    43.852 deg,	R =    54.361 deg
   GP2:
	UF : 1, UT : 1,
	J1=    90.000 deg,	J2=    90.000 deg
};
P[991]{
   GP1:
	UF : 1, UT : 1,		CONFIG : 'N U T, 0, 0, 0',
	X =  2458.273  mm,	Y =   -44.559  mm,	Z =   837.752  mm,
	W =    -1.320 deg,	P =    42.581 deg,	R =    55.585 deg
   GP2:
	UF : 1, UT : 1,
	J1=    90.000 deg,	J2=    90.000 deg
};
P[992]{
   GP1:
	UF : 1, UT : 1,		CONFIG : 'N U T, 0, 0, 0',
	X =  2655.577  mm,	Y =  -188.361  mm,	Z =   837.661  mm,
	W =   -30.971 deg,	P =    27.488 deg,	R =    12.662 deg
   GP2:
	UF : 1, UT : 1,
	J1=    90.000 deg,	J2=    90.000 deg
};
P[993]{
   GP1:
	UF : 1, UT : 1,		CONFIG : 'N U T, 0, 0, 0',
	X =  2658.956  mm,	Y =  -190.395  mm,	Z =   839.674  mm,
	W =   -30.965 deg,	P =    27.488 deg,	R =    12.663 deg
   GP2:
	UF : 1, UT : 1,
	J1=    90.000 deg,	J2=    90.000 deg
};
P[994]{
   GP1:
	UF : 1, UT : 1,		CONFIG : 'N U T, 0, 0, 0',
	X =  2073.431  mm,	Y =    50.699  mm,	Z =    17.153  mm,
	W =   -30.932 deg,	P =    -2.126 deg,	R =   142.465 deg
   GP2:
	UF : 1, UT : 1,
	J1=    80.000 deg,	J2=    90.000 deg
};
P[995]{
   GP1:
	UF : 1, UT : 1,		CONFIG : 'N U T, 0, 0, 0',
	X =  2111.468  mm,	Y =    13.622  mm,	Z =     7.245  mm,
	W =   -27.575 deg,	P =     5.122 deg,	R =   142.904 deg
   GP2:
	UF : 1, UT : 1,
	J1=    80.000 deg,	J2=    90.000 deg
};
P[996]{
   GP1:
	UF : 1, UT : 1,		CONFIG : 'N U T, 0, 0, 0',
	X =  2121.990  mm,	Y =     3.257  mm,	Z =     4.854  mm,
	W =   -27.571 deg,	P =     5.117 deg,	R =   139.585 deg
   GP2:
	UF : 1, UT : 1,
	J1=    80.000 deg,	J2=    90.000 deg
};
P[997]{
   GP1:
	UF : 1, UT : 1,		CONFIG : 'N U T, 0, 0, 0',
	X =  2127.968  mm,	Y =    -1.323  mm,	Z =     3.645  mm,
	W =   -27.577 deg,	P =     5.121 deg,	R =   136.987 deg
   GP2:
	UF : 1, UT : 1,
	J1=    80.000 deg,	J2=    90.000 deg
};
P[998]{
   GP1:
	UF : 1, UT : 1,		CONFIG : 'N U T, 0, 0, 0',
	X =  2250.493  mm,	Y =  -170.352  mm,	Z =   -14.380  mm,
	W =   -36.468 deg,	P =    -8.805 deg,	R =   122.587 deg
   GP2:
	UF : 1, UT : 1,
	J1=    80.000 deg,	J2=    90.000 deg
};
P[999]{
   GP1:
	UF : 1, UT : 1,		CONFIG : 'N U T, 0, 0, 0',
	X =  2258.054  mm,	Y =  -180.789  mm,	Z =   -16.004  mm,
	W =   -36.557 deg,	P =   -11.679 deg,	R =   125.980 deg
   GP2:
	UF : 1, UT : 1,
	J1=    80.000 deg,	J2=    90.000 deg
};
P[1000]{
   GP1:
	UF : 1, UT : 1,		CONFIG : 'N U T, 0, 0, 0',
	X =  2267.270  mm,	Y =  -192.246  mm,	Z =   -17.258  mm,
